SPLINE
SPL {X  -119.703, Y  +777.650, Z    +0.000, E1   -51.831, E3 +109843.279}
SPL {X  -145.184, Y  +738.720, Z    +0.000, E1   -43.488, E3 +109869.837}
SPL {X  -156.175, Y  +706.232, Z    +0.000, E1   -28.819, E3 +109878.722}
SPL {X  -159.337, Y  +685.942, Z    +0.000, E1   -14.672, E3 +109881.273}
SPL {X  -159.962, Y  +674.468, Z    +0.000, E1    -4.846, E3 +109881.892}
SPL {X  -159.990, Y  +669.479, Z    +0.000, E1    +0.004, E3 +109881.966}
SPL {X  -159.990, Y  +667.035, Z    +0.000, E1    +4.539, E3 +109881.997}
SPL {X  -159.990, Y  +662.914, Z    +0.000, E1   +13.494, E3 +109882.135}
SPL {X  -159.990, Y  +658.254, Z    +0.000, E1   +24.153, E3 +109882.413}
SPL {X  -159.990, Y  +652.944, Z    +0.000, E1   +35.122, E3 +109882.917}
SPL {X  -159.990, Y  +642.509, Z    +0.000, E1   +50.090, E3 +109884.488}
SPL {X  -159.990, Y  +618.566, Z    +0.000, E1   +64.119, E3 +109890.659}
SPL {X  -159.990, Y  +584.545, Z    +0.000, E1   +69.188, E3 +109903.194}
SPL {X  -159.990, Y  +578.002, Z    +0.000, E1   +69.607, E3 +109905.918}
SPL {X  -159.990, Y  +426.570, Z    +0.000, E1   +71.599, E3 +109986.408}
SPL {X  -159.990, Y  +405.946, Z    +0.000, E1   +71.630, E3 +110000.838}
SPL {X  -159.967, Y  +379.776, Z    +0.000, E1   +71.634, E3 +110019.284}
SPL {X  -158.535, Y  +360.970, Z    +0.000, E1   +71.460, E3 +110034.106}
SPL {X  -156.277, Y  +348.230, Z    +0.000, E1   +71.211, E3 +110045.450}
SPL {X  -155.351, Y  +344.251, Z    +0.000, E1   +70.004, E3 +110059.241}
SPL {X  -150.579, Y  +328.438, Z    +0.000, E1   +70.374, E3 +110067.627}
SPL {X  -146.933, Y  +319.195, Z    +0.000, E1   +70.230, E3 +110075.318}
SPL {X  -143.573, Y  +311.906, Z    +0.000, E1   +69.806, E3 +110083.628}
SPL {X  -139.693, Y  +304.508, Z    +0.000, E1   +69.301, E3 +110092.356}
SPL {X  -135.622, Y  +297.627, Z    +0.000, E1   +68.731, E3 +110100.764}
SPL {X  -131.165, Y  +290.889, Z    +0.000, E1   +68.094, E3 +110109.150}
SPL {X  -126.457, Y  +284.492, Z    +0.000, E1   +67.352, E3 +110117.235}
SPL {X  -123.432, Y  +280.710, Z    +0.000, E1   +66.830, E3 +110122.021}
SPL {X   -85.607, Y  +247.340, Z    +0.000, E1   +53.917, E3 +110263.742}
ENDSPLINE

SPLINE
SPL {X  -134.737, Y  +296.229, Z    +0.000, E1   +47.890, E3 +110406.515}
SPL {X  -154.917, Y  +342.531, Z    +0.000, E1   +31.203, E3 +110425.083}
SPL {X  -159.440, Y  +369.246, Z    +0.000, E1   +13.458, E3 +110428.982}
SPL {X  -159.987, Y  +381.470, Z    +0.000, E1    +2.976, E3 +110429.581}
SPL {X  -159.990, Y  +384.500, Z    +0.000, E1    +0.000, E3 +110429.614}
SPL {X  -159.990, Y  +386.323, Z    +0.000, E1    -3.079, E3 +110429.636}
SPL {X  -159.990, Y  +390.285, Z    +0.000, E1   -11.315, E3 +110429.757}
SPL {X  -159.990, Y  +394.559, Z    +0.000, E1   -20.770, E3 +110430.019}
SPL {X  -159.990, Y  +402.118, Z    +0.000, E1   -35.793, E3 +110430.810}
SPL {X  -159.990, Y  +415.193, Z    +0.000, E1   -52.724, E3 +110433.063}
SPL {X  -159.990, Y  +465.395, Z    +0.000, E1   -68.959, E3 +110448.152}
SPL {X  -159.990, Y  +657.157, Z    +0.000, E1   -72.499, E3 +110544.548}
SPL {X  -159.693, Y  +681.249, Z    +0.000, E1   -72.488, E3 +110560.942}
SPL {X  -157.599, Y  +699.059, Z    +0.000, E1   -72.249, E3 +110575.102}
SPL {X  -155.217, Y  +710.289, Z    +0.000, E1   -71.989, E3 +110585.119}
SPL {X  -152.611, Y  +719.527, Z    +0.000, E1   -71.702, E3 +110593.940}
SPL {X  -149.536, Y  +728.383, Z    +0.000, E1   -71.359, E3 +110602.919}
SPL {X  -146.250, Y  +736.367, Z    +0.000, E1   -70.965, E3 +110611.473}
SPL {X  -143.481, Y  +742.281, Z    +0.000, E1   -70.623, E3 +110618.069}
SPL {X  -140.071, Y  +748.811, Z    +0.000, E1   -70.193, E3 +110625.580}
SPL {X  -136.578, Y  +754.826, Z    +0.000, E1   -69.723, E3 +110632.710}
SPL {X  -133.265, Y  +760.028, Z    +0.000, E1   -69.258, E3 +110639.011}
SPL {X  -129.890, Y  +764.909, Z    +0.000, E1   -68.775, E3 +110644.981}
SPL {X  -125.802, Y  +770.346, Z    +0.000, E1   -68.156, E3 +110651.681}
SPL {X  -122.624, Y  +774.263, Z    +0.000, E1   -67.622, E3 +110656.503}
SPL {X   -84.435, Y  +807.395, Z    +0.000, E1   -55.948, E3 +110767.508}
ENDSPLINE

SPLINE
SPL {X  -119.703, Y  +777.650, Z    +0.000, E1   -51.831, E3 +110931.514}
SPL {X  -145.184, Y  +738.720, Z    +0.000, E1   -43.488, E3 +110958.072}
SPL {X  -154.467, Y  +713.173, Z    +0.000, E1   -32.658, E3 +110965.668}
SPL {X  -157.530, Y  +699.446, Z    +0.000, E1   -24.482, E3 +110968.084}
SPL {X  -159.337, Y  +685.942, Z    +0.000, E1   -14.672, E3 +110969.508}
SPL {X  -159.962, Y  +674.468, Z    +0.000, E1    -4.846, E3 +110970.127}
SPL {X  -159.990, Y  +669.479, Z    +0.000, E1    +0.004, E3 +110970.201}
SPL {X  -159.990, Y  +667.035, Z    +0.000, E1    +4.539, E3 +110970.232}
SPL {X  -159.990, Y  +662.914, Z    +0.000, E1   +13.494, E3 +110970.371}
SPL {X  -159.990, Y  +658.254, Z    +0.000, E1   +24.153, E3 +110970.648}
SPL {X  -159.990, Y  +652.944, Z    +0.000, E1   +35.122, E3 +110971.152}
SPL {X  -159.990, Y  +642.509, Z    +0.000, E1   +50.090, E3 +110972.724}
SPL {X  -159.990, Y  +618.566, Z    +0.000, E1   +64.119, E3 +110978.894}
SPL {X  -159.990, Y  +582.261, Z    +0.000, E1   +69.343, E3 +110992.380}
SPL {X  -159.990, Y  +406.555, Z    +0.000, E1   +71.635, E3 +111088.627}
SPL {X  -159.967, Y  +379.776, Z    +0.000, E1   +71.634, E3 +111107.520}
SPL {X  -158.535, Y  +360.970, Z    +0.000, E1   +71.460, E3 +111122.342}
SPL {X  -156.882, Y  +351.118, Z    +0.000, E1   +71.263, E3 +111131.053}
SPL {X  -155.538, Y  +345.018, Z    +0.000, E1   +71.109, E3 +111136.760}
SPL {X  -155.351, Y  +344.251, Z    +0.000, E1   +70.004, E3 +111147.477}
SPL {X  -150.579, Y  +328.438, Z    +0.000, E1   +70.374, E3 +111155.862}
SPL {X  -146.933, Y  +319.195, Z    +0.000, E1   +70.230, E3 +111163.553}
SPL {X  -143.573, Y  +311.906, Z    +0.000, E1   +69.806, E3 +111171.863}
SPL {X  -140.547, Y  +306.057, Z    +0.000, E1   +69.399, E3 +111178.755}
SPL {X  -137.438, Y  +300.600, Z    +0.000, E1   +68.984, E3 +111185.350}
SPL {X  -133.397, Y  +294.172, Z    +0.000, E1   +68.416, E3 +111193.285}
SPL {X  -128.822, Y  +287.623, Z    +0.000, E1   +67.729, E3 +111201.509}
SPL {X  -124.502, Y  +282.021, Z    +0.000, E1   +67.035, E3 +111208.583}
SPL {X   -85.607, Y  +247.340, Z    +0.000, E1   +53.917, E3 +111351.978}
ENDSPLINE

SPLINE
SPL {X  -134.737, Y  +296.229, Z    +0.000, E1   +47.890, E3 +111494.750}
SPL {X  -154.917, Y  +342.531, Z    +0.000, E1   +31.203, E3 +111513.318}
SPL {X  -159.440, Y  +369.246, Z    +0.000, E1   +13.458, E3 +111517.217}
SPL {X  -159.957, Y  +379.264, Z    +0.000, E1    +4.909, E3 +111517.773}
SPL {X  -159.990, Y  +384.398, Z    +0.000, E1    +0.172, E3 +111517.849}
SPL {X  -159.990, Y  +386.323, Z    +0.000, E1    -3.079, E3 +111517.871}
SPL {X  -159.990, Y  +390.285, Z    +0.000, E1   -11.315, E3 +111517.992}
SPL {X  -159.990, Y  +394.559, Z    +0.000, E1   -20.770, E3 +111518.254}
SPL {X  -159.990, Y  +402.118, Z    +0.000, E1   -35.793, E3 +111519.046}
SPL {X  -159.990, Y  +415.193, Z    +0.000, E1   -52.724, E3 +111521.298}
SPL {X  -159.990, Y  +465.395, Z    +0.000, E1   -68.959, E3 +111536.387}
SPL {X  -159.990, Y  +657.157, Z    +0.000, E1   -72.499, E3 +111632.784}
SPL {X  -159.947, Y  +675.227, Z    +0.000, E1   -72.487, E3 +111644.944}
SPL {X  -159.251, Y  +686.856, Z    +0.000, E1   -72.412, E3 +111653.472}
SPL {X  -157.599, Y  +699.059, Z    +0.000, E1   -72.249, E3 +111663.337}
SPL {X  -155.217, Y  +710.289, Z    +0.000, E1   -71.989, E3 +111673.354}
SPL {X  -152.611, Y  +719.527, Z    +0.000, E1   -71.702, E3 +111682.175}
SPL {X  -149.536, Y  +728.383, Z    +0.000, E1   -71.359, E3 +111691.154}
SPL {X  -146.250, Y  +736.367, Z    +0.000, E1   -70.965, E3 +111699.709}
SPL {X  -143.481, Y  +742.281, Z    +0.000, E1   -70.623, E3 +111706.304}
SPL {X  -140.071, Y  +748.811, Z    +0.000, E1   -70.193, E3 +111713.816}
SPL {X  -136.578, Y  +754.826, Z    +0.000, E1   -69.723, E3 +111720.945}
SPL {X  -133.265, Y  +760.028, Z    +0.000, E1   -69.258, E3 +111727.246}
SPL {X  -130.837, Y  +763.579, Z    +0.000, E1   -68.898, E3 +111731.606}
SPL {X  -127.941, Y  +767.561, Z    +0.000, E1   -68.475, E3 +111736.496}
SPL {X  -123.778, Y  +772.869, Z    +0.000, E1   -67.843, E3 +111743.004}
SPL {X   -84.435, Y  +807.395, Z    +0.000, E1   -55.948, E3 +111855.743}
ENDSPLINE

SPLINE
SPL {X  -119.703, Y  +777.650, Z    +0.000, E1   -51.831, E3 +112019.750}
SPL {X  -145.184, Y  +738.720, Z    +0.000, E1   -43.488, E3 +112046.308}
SPL {X  -154.467, Y  +713.173, Z    +0.000, E1   -32.658, E3 +112053.903}
SPL {X  -157.530, Y  +699.446, Z    +0.000, E1   -24.482, E3 +112056.319}
SPL {X  -159.337, Y  +685.942, Z    +0.000, E1   -14.672, E3 +112057.744}
SPL {X  -159.962, Y  +674.468, Z    +0.000, E1    -4.846, E3 +112058.362}
SPL {X  -159.990, Y  +669.479, Z    +0.000, E1    +0.004, E3 +112058.436}
SPL {X  -159.990, Y  +667.035, Z    +0.000, E1    +4.539, E3 +112058.467}
SPL {X  -159.990, Y  +662.914, Z    +0.000, E1   +13.494, E3 +112058.606}
SPL {X  -159.990, Y  +658.254, Z    +0.000, E1   +24.153, E3 +112058.884}
SPL {X  -159.990, Y  +652.944, Z    +0.000, E1   +35.122, E3 +112059.387}
SPL {X  -159.990, Y  +642.509, Z    +0.000, E1   +50.090, E3 +112060.959}
SPL {X  -159.990, Y  +618.566, Z    +0.000, E1   +64.119, E3 +112067.130}
SPL {X  -159.990, Y  +582.261, Z    +0.000, E1   +69.343, E3 +112080.615}
SPL {X  -159.990, Y  +406.555, Z    +0.000, E1   +71.635, E3 +112176.862}
SPL {X  -159.990, Y  +385.723, Z    +0.000, E1   +71.610, E3 +112191.600}
SPL {X  -159.404, Y  +368.814, Z    +0.000, E1   +71.556, E3 +112204.129}
SPL {X  -158.061, Y  +357.731, Z    +0.000, E1   +71.393, E3 +112213.397}
SPL {X  -156.277, Y  +348.230, Z    +0.000, E1   +71.211, E3 +112221.920}
SPL {X  -155.351, Y  +344.251, Z    +0.000, E1   +70.004, E3 +112235.712}
SPL {X  -150.579, Y  +328.438, Z    +0.000, E1   +70.374, E3 +112244.097}
SPL {X  -146.933, Y  +319.195, Z    +0.000, E1   +70.230, E3 +112251.788}
SPL {X  -143.573, Y  +311.906, Z    +0.000, E1   +69.806, E3 +112260.099}
SPL {X  -140.547, Y  +306.057, Z    +0.000, E1   +69.399, E3 +112266.991}
SPL {X  -137.438, Y  +300.600, Z    +0.000, E1   +68.984, E3 +112273.585}
SPL {X  -133.397, Y  +294.172, Z    +0.000, E1   +68.416, E3 +112281.520}
SPL {X  -128.822, Y  +287.623, Z    +0.000, E1   +67.729, E3 +112289.744}
SPL {X  -124.502, Y  +282.021, Z    +0.000, E1   +67.035, E3 +112296.818}
SPL {X   -85.607, Y  +247.340, Z    +0.000, E1   +53.917, E3 +112440.213}
ENDSPLINE

SPLINE
SPL {X  -134.737, Y  +296.229, Z    +0.000, E1   +47.890, E3 +112582.986}
SPL {X  -153.211, Y  +336.421, Z    +0.000, E1   +34.262, E3 +112600.194}
SPL {X  -158.240, Y  +358.900, Z    +0.000, E1   +21.089, E3 +112604.399}
SPL {X  -159.674, Y  +372.451, Z    +0.000, E1   +10.778, E3 +112605.695}
SPL {X  -159.987, Y  +381.470, Z    +0.000, E1    +2.976, E3 +112606.052}
SPL {X  -159.990, Y  +384.761, Z    +0.000, E1    -0.257, E3 +112606.087}
SPL {X  -159.990, Y  +389.248, Z    +0.000, E1    -8.879, E3 +112606.191}
SPL {X  -159.990, Y  +394.559, Z    +0.000, E1   -20.770, E3 +112606.490}
SPL {X  -159.990, Y  +402.118, Z    +0.000, E1   -35.793, E3 +112607.281}
SPL {X  -159.990, Y  +415.193, Z    +0.000, E1   -52.724, E3 +112609.534}
SPL {X  -159.990, Y  +465.395, Z    +0.000, E1   -68.959, E3 +112624.622}
SPL {X  -159.990, Y  +657.157, Z    +0.000, E1   -72.499, E3 +112721.019}
SPL {X  -159.693, Y  +681.249, Z    +0.000, E1   -72.488, E3 +112737.413}
SPL {X  -157.599, Y  +699.059, Z    +0.000, E1   -72.249, E3 +112751.573}
SPL {X  -155.217, Y  +710.289, Z    +0.000, E1   -71.989, E3 +112761.589}
SPL {X  -152.611, Y  +719.527, Z    +0.000, E1   -71.702, E3 +112770.410}
SPL {X  -149.536, Y  +728.383, Z    +0.000, E1   -71.359, E3 +112779.390}
SPL {X  -146.250, Y  +736.367, Z    +0.000, E1   -70.965, E3 +112787.944}
SPL {X  -143.481, Y  +742.281, Z    +0.000, E1   -70.623, E3 +112794.539}
SPL {X  -140.071, Y  +748.811, Z    +0.000, E1   -70.193, E3 +112802.051}
SPL {X  -136.578, Y  +754.826, Z    +0.000, E1   -69.723, E3 +112809.180}
SPL {X  -133.265, Y  +760.028, Z    +0.000, E1   -69.258, E3 +112815.481}
SPL {X  -130.837, Y  +763.579, Z    +0.000, E1   -68.898, E3 +112819.841}
SPL {X  -127.941, Y  +767.561, Z    +0.000, E1   -68.475, E3 +112824.732}
SPL {X  -123.778, Y  +772.869, Z    +0.000, E1   -67.843, E3 +112831.239}
SPL {X   -84.435, Y  +807.395, Z    +0.000, E1   -55.948, E3 +112943.978}
ENDSPLINE

SPLINE
SPL {X  -119.703, Y  +777.650, Z    +0.000, E1   -51.831, E3 +113107.985}
SPL {X  -145.184, Y  +738.720, Z    +0.000, E1   -43.488, E3 +113134.543}
SPL {X  -156.175, Y  +706.232, Z    +0.000, E1   -28.819, E3 +113143.428}
SPL {X  -159.337, Y  +685.942, Z    +0.000, E1   -14.672, E3 +113145.979}
SPL {X  -159.900, Y  +676.871, Z    +0.000, E1    -6.955, E3 +113146.527}
SPL {X  -159.990, Y  +669.634, Z    +0.000, E1    -0.285, E3 +113146.670}
SPL {X  -159.990, Y  +667.035, Z    +0.000, E1    +4.539, E3 +113146.702}
SPL {X  -159.990, Y  +662.914, Z    +0.000, E1   +13.494, E3 +113146.841}
SPL {X  -159.990, Y  +658.254, Z    +0.000, E1   +24.153, E3 +113147.119}
SPL {X  -159.990, Y  +652.944, Z    +0.000, E1   +35.122, E3 +113147.623}
SPL {X  -159.990, Y  +642.509, Z    +0.000, E1   +50.090, E3 +113149.194}
SPL {X  -159.990, Y  +618.566, Z    +0.000, E1   +64.119, E3 +113155.365}
SPL {X  -159.990, Y  +584.545, Z    +0.000, E1   +69.188, E3 +113167.900}
SPL {X  -159.990, Y  +578.002, Z    +0.000, E1   +69.607, E3 +113170.624}
SPL {X  -159.990, Y  +426.570, Z    +0.000, E1   +71.599, E3 +113251.114}
SPL {X  -159.990, Y  +405.946, Z    +0.000, E1   +71.630, E3 +113265.544}
SPL {X  -159.967, Y  +379.776, Z    +0.000, E1   +71.634, E3 +113283.990}
SPL {X  -158.535, Y  +360.970, Z    +0.000, E1   +71.460, E3 +113298.812}
SPL {X  -156.277, Y  +348.230, Z    +0.000, E1   +71.211, E3 +113310.155}
SPL {X  -155.351, Y  +344.251, Z    +0.000, E1   +70.004, E3 +113323.947}
SPL {X  -150.579, Y  +328.438, Z    +0.000, E1   +70.374, E3 +113332.333}
SPL {X  -146.933, Y  +319.195, Z    +0.000, E1   +70.230, E3 +113340.024}
SPL {X  -143.573, Y  +311.906, Z    +0.000, E1   +69.806, E3 +113348.334}
SPL {X  -140.547, Y  +306.057, Z    +0.000, E1   +69.399, E3 +113355.226}
SPL {X  -137.438, Y  +300.600, Z    +0.000, E1   +68.984, E3 +113361.820}
SPL {X  -133.397, Y  +294.172, Z    +0.000, E1   +68.416, E3 +113369.755}
SPL {X  -129.981, Y  +289.217, Z    +0.000, E1   +67.880, E3 +113376.005}
SPL {X  -126.457, Y  +284.492, Z    +0.000, E1   +67.352, E3 +113381.941}
SPL {X  -123.432, Y  +280.710, Z    +0.000, E1   +66.830, E3 +113386.727}
SPL {X   -85.607, Y  +247.340, Z    +0.000, E1   +53.917, E3 +113528.448}
ENDSPLINE

SPLINE
SPL {X  -119.557, Y  +276.184, Z    +0.000, E1   +51.032, E3 +113651.985}
SPL {X  -138.294, Y  +302.054, Z    +0.000, E1   +46.576, E3 +113675.307}
SPL {X  -153.211, Y  +336.421, Z    +0.000, E1   +34.262, E3 +113688.429}
SPL {X  -158.240, Y  +358.900, Z    +0.000, E1   +21.089, E3 +113692.634}
SPL {X  -159.854, Y  +375.896, Z    +0.000, E1    +7.981, E3 +113694.100}
SPL {X  -159.990, Y  +384.398, Z    +0.000, E1    +0.172, E3 +113694.320}
SPL {X  -159.990, Y  +386.323, Z    +0.000, E1    -3.079, E3 +113694.342}
SPL {X  -159.990, Y  +390.285, Z    +0.000, E1   -11.315, E3 +113694.463}
SPL {X  -159.990, Y  +394.559, Z    +0.000, E1   -20.770, E3 +113694.725}
SPL {X  -159.990, Y  +402.118, Z    +0.000, E1   -35.793, E3 +113695.516}
SPL {X  -159.990, Y  +415.193, Z    +0.000, E1   -52.724, E3 +113697.769}
SPL {X  -159.990, Y  +465.395, Z    +0.000, E1   -68.959, E3 +113712.857}
SPL {X  -159.990, Y  +657.157, Z    +0.000, E1   -72.499, E3 +113809.254}
SPL {X  -159.693, Y  +681.249, Z    +0.000, E1   -72.488, E3 +113825.648}
SPL {X  -157.599, Y  +699.059, Z    +0.000, E1   -72.249, E3 +113839.808}
SPL {X  -155.217, Y  +710.289, Z    +0.000, E1   -71.989, E3 +113849.825}
SPL {X  -152.611, Y  +719.527, Z    +0.000, E1   -71.702, E3 +113858.646}
SPL {X  -149.536, Y  +728.383, Z    +0.000, E1   -71.359, E3 +113867.625}
SPL {X  -146.250, Y  +736.367, Z    +0.000, E1   -70.965, E3 +113876.179}
SPL {X  -143.481, Y  +742.281, Z    +0.000, E1   -70.623, E3 +113882.775}
SPL {X  -140.071, Y  +748.811, Z    +0.000, E1   -70.193, E3 +113890.286}
SPL {X  -136.578, Y  +754.826, Z    +0.000, E1   -69.723, E3 +113897.416}
SPL {X  -133.265, Y  +760.028, Z    +0.000, E1   -69.258, E3 +113903.717}
SPL {X  -129.890, Y  +764.909, Z    +0.000, E1   -68.775, E3 +113909.687}
SPL {X  -125.802, Y  +770.346, Z    +0.000, E1   -68.156, E3 +113916.386}
SPL {X  -122.624, Y  +774.263, Z    +0.000, E1   -67.622, E3 +113921.209}
SPL {X   -84.435, Y  +807.395, Z    +0.000, E1   -55.948, E3 +114032.214}
ENDSPLINE

SPLINE
SPL {X  -119.703, Y  +777.650, Z    +0.000, E1   -51.831, E3 +114196.220}
SPL {X  -145.184, Y  +738.720, Z    +0.000, E1   -43.488, E3 +114222.778}
SPL {X  -154.467, Y  +713.173, Z    +0.000, E1   -32.658, E3 +114230.374}
SPL {X  -157.530, Y  +699.446, Z    +0.000, E1   -24.482, E3 +114232.789}
SPL {X  -159.337, Y  +685.942, Z    +0.000, E1   -14.672, E3 +114234.214}
SPL {X  -159.900, Y  +676.871, Z    +0.000, E1    -6.955, E3 +114234.762}
SPL {X  -159.990, Y  +669.634, Z    +0.000, E1    -0.285, E3 +114234.906}
SPL {X  -159.990, Y  +667.035, Z    +0.000, E1    +4.539, E3 +114234.938}
SPL {X  -159.990, Y  +662.914, Z    +0.000, E1   +13.494, E3 +114235.077}
SPL {X  -159.990, Y  +658.254, Z    +0.000, E1   +24.153, E3 +114235.354}
SPL {X  -159.990, Y  +650.381, Z    +0.000, E1   +39.393, E3 +114236.206}
SPL {X  -159.990, Y  +638.701, Z    +0.000, E1   +53.953, E3 +114238.092}
SPL {X  -159.990, Y  +618.566, Z    +0.000, E1   +64.119, E3 +114243.600}
SPL {X  -159.990, Y  +582.261, Z    +0.000, E1   +69.343, E3 +114257.086}
SPL {X  -159.990, Y  +406.555, Z    +0.000, E1   +71.635, E3 +114353.332}
SPL {X  -159.990, Y  +385.723, Z    +0.000, E1   +71.610, E3 +114368.071}
SPL {X  -159.404, Y  +368.814, Z    +0.000, E1   +71.556, E3 +114380.600}
SPL {X  -158.061, Y  +357.731, Z    +0.000, E1   +71.393, E3 +114389.868}
SPL {X  -156.277, Y  +348.230, Z    +0.000, E1   +71.211, E3 +114398.391}
SPL {X  -155.351, Y  +344.251, Z    +0.000, E1   +70.004, E3 +114412.183}
SPL {X  -150.579, Y  +328.438, Z    +0.000, E1   +70.374, E3 +114420.568}
SPL {X  -146.933, Y  +319.195, Z    +0.000, E1   +70.230, E3 +114428.259}
SPL {X  -143.573, Y  +311.906, Z    +0.000, E1   +69.806, E3 +114436.569}
SPL {X  -140.547, Y  +306.057, Z    +0.000, E1   +69.399, E3 +114443.461}
SPL {X  -137.438, Y  +300.600, Z    +0.000, E1   +68.984, E3 +114450.056}
SPL {X  -133.397, Y  +294.172, Z    +0.000, E1   +68.416, E3 +114457.990}
SPL {X  -128.822, Y  +287.623, Z    +0.000, E1   +67.729, E3 +114466.215}
SPL {X  -124.502, Y  +282.021, Z    +0.000, E1   +67.035, E3 +114473.289}
SPL {X   -85.607, Y  +247.340, Z    +0.000, E1   +53.917, E3 +114616.683}
ENDSPLINE

SPLINE
SPL {X  -134.737, Y  +296.229, Z    +0.000, E1   +47.890, E3 +114759.456}
SPL {X  -154.917, Y  +342.531, Z    +0.000, E1   +31.203, E3 +114778.024}
SPL {X  -159.440, Y  +369.246, Z    +0.000, E1   +13.458, E3 +114781.923}
SPL {X  -159.987, Y  +381.470, Z    +0.000, E1    +2.976, E3 +114782.522}
SPL {X  -159.990, Y  +384.500, Z    +0.000, E1    +0.000, E3 +114782.555}
SPL {X  -159.990, Y  +386.323, Z    +0.000, E1    -3.079, E3 +114782.577}
SPL {X  -159.990, Y  +390.285, Z    +0.000, E1   -11.315, E3 +114782.698}
SPL {X  -159.990, Y  +394.559, Z    +0.000, E1   -20.770, E3 +114782.960}
SPL {X  -159.990, Y  +399.334, Z    +0.000, E1   -30.876, E3 +114783.399}
SPL {X  -159.990, Y  +405.006, Z    +0.000, E1   -40.810, E3 +114784.117}
SPL {X  -159.990, Y  +415.193, Z    +0.000, E1   -52.724, E3 +114786.004}
SPL {X  -159.990, Y  +465.395, Z    +0.000, E1   -68.959, E3 +114801.093}
SPL {X  -159.990, Y  +657.157, Z    +0.000, E1   -72.499, E3 +114897.490}
SPL {X  -159.693, Y  +681.249, Z    +0.000, E1   -72.488, E3 +114913.884}
SPL {X  -157.599, Y  +699.059, Z    +0.000, E1   -72.249, E3 +114928.043}
SPL {X  -155.217, Y  +710.289, Z    +0.000, E1   -71.989, E3 +114938.060}
SPL {X  -152.611, Y  +719.527, Z    +0.000, E1   -71.702, E3 +114946.881}
SPL {X  -149.536, Y  +728.383, Z    +0.000, E1   -71.359, E3 +114955.860}
SPL {X  -146.250, Y  +736.367, Z    +0.000, E1   -70.965, E3 +114964.414}
SPL {X  -143.481, Y  +742.281, Z    +0.000, E1   -70.623, E3 +114971.010}
SPL {X  -140.071, Y  +748.811, Z    +0.000, E1   -70.193, E3 +114978.522}
SPL {X  -136.578, Y  +754.826, Z    +0.000, E1   -69.723, E3 +114985.651}
SPL {X  -133.265, Y  +760.028, Z    +0.000, E1   -69.258, E3 +114991.952}
SPL {X  -130.837, Y  +763.579, Z    +0.000, E1   -68.898, E3 +114996.312}
SPL {X  -127.941, Y  +767.561, Z    +0.000, E1   -68.475, E3 +115001.202}
SPL {X  -123.778, Y  +772.869, Z    +0.000, E1   -67.843, E3 +115007.710}
SPL {X   -84.435, Y  +807.395, Z    +0.000, E1   -55.948, E3 +115120.449}
ENDSPLINE

SPLINE
SPL {X  -119.703, Y  +777.650, Z    +0.000, E1   -51.831, E3 +115284.455}
SPL {X  -145.184, Y  +738.720, Z    +0.000, E1   -43.488, E3 +115311.013}
SPL {X  -156.175, Y  +706.232, Z    +0.000, E1   -28.819, E3 +115319.898}
SPL {X  -159.337, Y  +685.942, Z    +0.000, E1   -14.672, E3 +115322.449}
SPL {X  -159.962, Y  +674.468, Z    +0.000, E1    -4.846, E3 +115323.068}
SPL {X  -159.990, Y  +669.479, Z    +0.000, E1    +0.004, E3 +115323.142}
SPL {X  -159.990, Y  +667.035, Z    +0.000, E1    +4.539, E3 +115323.173}
SPL {X  -159.990, Y  +662.914, Z    +0.000, E1   +13.494, E3 +115323.312}
SPL {X  -159.990, Y  +658.254, Z    +0.000, E1   +24.153, E3 +115323.590}
SPL {X  -159.990, Y  +652.944, Z    +0.000, E1   +35.122, E3 +115324.093}
SPL {X  -159.990, Y  +642.509, Z    +0.000, E1   +50.090, E3 +115325.665}
SPL {X  -159.990, Y  +618.566, Z    +0.000, E1   +64.119, E3 +115331.835}
SPL {X  -159.990, Y  +584.545, Z    +0.000, E1   +69.188, E3 +115344.371}
SPL {X  -159.990, Y  +578.002, Z    +0.000, E1   +69.607, E3 +115347.094}
SPL {X  -159.990, Y  +426.570, Z    +0.000, E1   +71.599, E3 +115427.584}
SPL {X  -159.990, Y  +405.946, Z    +0.000, E1   +71.630, E3 +115442.014}
SPL {X  -159.967, Y  +379.776, Z    +0.000, E1   +71.634, E3 +115460.461}
SPL {X  -158.535, Y  +360.970, Z    +0.000, E1   +71.460, E3 +115475.283}
SPL {X  -156.882, Y  +351.118, Z    +0.000, E1   +71.263, E3 +115483.995}
SPL {X  -155.889, Y  +346.508, Z    +0.000, E1   +70.461, E3 +115494.857}
SPL {X  -154.332, Y  +340.328, Z    +0.000, E1   +70.024, E3 +115503.085}
SPL {X  -150.579, Y  +328.438, Z    +0.000, E1   +70.374, E3 +115508.803}
SPL {X  -146.933, Y  +319.195, Z    +0.000, E1   +70.230, E3 +115516.494}
SPL {X  -143.573, Y  +311.906, Z    +0.000, E1   +69.806, E3 +115524.805}
SPL {X  -139.693, Y  +304.508, Z    +0.000, E1   +69.301, E3 +115533.533}
SPL {X  -135.622, Y  +297.627, Z    +0.000, E1   +68.731, E3 +115541.941}
SPL {X  -131.165, Y  +290.889, Z    +0.000, E1   +68.094, E3 +115550.326}
SPL {X  -126.457, Y  +284.492, Z    +0.000, E1   +67.352, E3 +115558.412}
SPL {X  -123.432, Y  +280.710, Z    +0.000, E1   +66.830, E3 +115563.197}
SPL {X   -85.607, Y  +247.340, Z    +0.000, E1   +53.917, E3 +115704.919}
ENDSPLINE

SPLINE
SPL {X  -134.737, Y  +296.229, Z    +0.000, E1   +47.890, E3 +115847.692}
SPL {X  -154.917, Y  +342.531, Z    +0.000, E1   +31.203, E3 +115866.259}
SPL {X  -159.440, Y  +369.246, Z    +0.000, E1   +13.458, E3 +115870.159}
SPL {X  -159.987, Y  +381.470, Z    +0.000, E1    +2.976, E3 +115870.757}
SPL {X  -159.990, Y  +384.500, Z    +0.000, E1    +0.000, E3 +115870.791}
SPL {X  -159.990, Y  +386.323, Z    +0.000, E1    -3.079, E3 +115870.812}
SPL {X  -159.990, Y  +390.285, Z    +0.000, E1   -11.315, E3 +115870.933}
SPL {X  -159.990, Y  +394.559, Z    +0.000, E1   -20.770, E3 +115871.195}
SPL {X  -159.990, Y  +399.334, Z    +0.000, E1   -30.876, E3 +115871.634}
SPL {X  -159.990, Y  +405.006, Z    +0.000, E1   -40.810, E3 +115872.352}
SPL {X  -159.990, Y  +415.193, Z    +0.000, E1   -52.724, E3 +115874.239}
SPL {X  -159.990, Y  +465.395, Z    +0.000, E1   -68.959, E3 +115889.328}
SPL {X  -159.990, Y  +657.157, Z    +0.000, E1   -72.499, E3 +115985.725}
SPL {X  -159.693, Y  +681.249, Z    +0.000, E1   -72.488, E3 +116002.119}
SPL {X  -157.599, Y  +699.059, Z    +0.000, E1   -72.249, E3 +116016.278}
SPL {X  -155.217, Y  +710.289, Z    +0.000, E1   -71.989, E3 +116026.295}
SPL {X  -152.611, Y  +719.527, Z    +0.000, E1   -71.702, E3 +116035.116}
SPL {X  -149.536, Y  +728.383, Z    +0.000, E1   -71.359, E3 +116044.096}
SPL {X  -146.250, Y  +736.367, Z    +0.000, E1   -70.965, E3 +116052.650}
SPL {X  -143.481, Y  +742.281, Z    +0.000, E1   -70.623, E3 +116059.245}
SPL {X  -140.071, Y  +748.811, Z    +0.000, E1   -70.193, E3 +116066.757}
SPL {X  -136.578, Y  +754.826, Z    +0.000, E1   -69.723, E3 +116073.886}
SPL {X  -133.265, Y  +760.028, Z    +0.000, E1   -69.258, E3 +116080.187}
SPL {X  -130.837, Y  +763.579, Z    +0.000, E1   -68.898, E3 +116084.547}
SPL {X  -127.941, Y  +767.561, Z    +0.000, E1   -68.475, E3 +116089.438}
SPL {X  -123.778, Y  +772.869, Z    +0.000, E1   -67.843, E3 +116095.945}
SPL {X   -84.435, Y  +807.395, Z    +0.000, E1   -55.948, E3 +116208.684}
ENDSPLINE

SPLINE
SPL {X  -119.703, Y  +777.650, Z    +0.000, E1   -51.831, E3 +116372.691}
SPL {X  -145.184, Y  +738.720, Z    +0.000, E1   -43.488, E3 +116399.249}
SPL {X  -156.175, Y  +706.232, Z    +0.000, E1   -28.819, E3 +116408.134}
SPL {X  -159.337, Y  +685.942, Z    +0.000, E1   -14.672, E3 +116410.685}
SPL {X  -159.962, Y  +674.468, Z    +0.000, E1    -4.846, E3 +116411.303}
SPL {X  -159.990, Y  +669.479, Z    +0.000, E1    +0.004, E3 +116411.378}
SPL {X  -159.990, Y  +667.035, Z    +0.000, E1    +4.539, E3 +116411.408}
SPL {X  -159.990, Y  +662.914, Z    +0.000, E1   +13.494, E3 +116411.547}
SPL {X  -159.990, Y  +658.254, Z    +0.000, E1   +24.153, E3 +116411.825}
SPL {X  -159.990, Y  +652.944, Z    +0.000, E1   +35.122, E3 +116412.329}
SPL {X  -159.990, Y  +646.557, Z    +0.000, E1   +45.390, E3 +116413.195}
SPL {X  -159.990, Y  +638.701, Z    +0.000, E1   +53.953, E3 +116414.562}
SPL {X  -159.990, Y  +618.566, Z    +0.000, E1   +64.119, E3 +116420.071}
SPL {X  -159.990, Y  +582.261, Z    +0.000, E1   +69.343, E3 +116433.556}
SPL {X  -159.990, Y  +426.570, Z    +0.000, E1   +71.599, E3 +116515.820}
SPL {X  -159.990, Y  +405.946, Z    +0.000, E1   +71.630, E3 +116530.250}
SPL {X  -159.990, Y  +385.723, Z    +0.000, E1   +71.610, E3 +116544.541}
SPL {X  -159.404, Y  +368.814, Z    +0.000, E1   +71.556, E3 +116557.071}
SPL {X  -158.061, Y  +357.731, Z    +0.000, E1   +71.393, E3 +116566.338}
SPL {X  -156.277, Y  +348.230, Z    +0.000, E1   +71.211, E3 +116574.861}
SPL {X  -155.351, Y  +344.251, Z    +0.000, E1   +70.004, E3 +116588.653}
SPL {X  -150.579, Y  +328.438, Z    +0.000, E1   +70.374, E3 +116597.039}
SPL {X  -146.933, Y  +319.195, Z    +0.000, E1   +70.230, E3 +116604.730}
SPL {X  -143.573, Y  +311.906, Z    +0.000, E1   +69.806, E3 +116613.040}
SPL {X  -140.547, Y  +306.057, Z    +0.000, E1   +69.399, E3 +116619.932}
SPL {X  -136.400, Y  +298.883, Z    +0.000, E1   +68.867, E3 +116628.588}
SPL {X  -131.165, Y  +290.889, Z    +0.000, E1   +68.094, E3 +116638.562}
SPL {X  -126.457, Y  +284.492, Z    +0.000, E1   +67.352, E3 +116646.647}
SPL {X  -123.432, Y  +280.710, Z    +0.000, E1   +66.830, E3 +116651.433}
SPL {X   -85.607, Y  +247.340, Z    +0.000, E1   +53.917, E3 +116793.154}
ENDSPLINE

SPLINE
SPL {X  -119.557, Y  +276.184, Z    +0.000, E1   +51.032, E3 +116916.691}
SPL {X  -138.294, Y  +302.054, Z    +0.000, E1   +46.576, E3 +116940.013}
SPL {X  -153.211, Y  +336.421, Z    +0.000, E1   +34.262, E3 +116953.135}
SPL {X  -158.240, Y  +358.900, Z    +0.000, E1   +21.089, E3 +116957.340}
SPL {X  -159.674, Y  +372.451, Z    +0.000, E1   +10.778, E3 +116958.636}
SPL {X  -159.987, Y  +381.470, Z    +0.000, E1    +2.976, E3 +116958.993}
SPL {X  -159.990, Y  +384.761, Z    +0.000, E1    -0.257, E3 +116959.028}
SPL {X  -159.990, Y  +389.248, Z    +0.000, E1    -8.879, E3 +116959.132}
SPL {X  -159.990, Y  +394.559, Z    +0.000, E1   -20.770, E3 +116959.431}
SPL {X  -159.990, Y  +402.118, Z    +0.000, E1   -35.793, E3 +116960.222}
SPL {X  -159.990, Y  +415.193, Z    +0.000, E1   -52.724, E3 +116962.475}
SPL {X  -159.990, Y  +465.395, Z    +0.000, E1   -68.959, E3 +116977.563}
SPL {X  -159.990, Y  +657.157, Z    +0.000, E1   -72.499, E3 +117073.960}
SPL {X  -159.947, Y  +675.227, Z    +0.000, E1   -72.487, E3 +117086.120}
SPL {X  -159.251, Y  +686.856, Z    +0.000, E1   -72.412, E3 +117094.648}
SPL {X  -157.599, Y  +699.059, Z    +0.000, E1   -72.249, E3 +117104.514}
SPL {X  -155.217, Y  +710.289, Z    +0.000, E1   -71.989, E3 +117114.530}
SPL {X  -152.611, Y  +719.527, Z    +0.000, E1   -71.702, E3 +117123.352}
SPL {X  -149.536, Y  +728.383, Z    +0.000, E1   -71.359, E3 +117132.331}
SPL {X  -146.250, Y  +736.367, Z    +0.000, E1   -70.965, E3 +117140.885}
SPL {X  -143.481, Y  +742.281, Z    +0.000, E1   -70.623, E3 +117147.480}
SPL {X  -140.071, Y  +748.811, Z    +0.000, E1   -70.193, E3 +117154.992}
SPL {X  -136.578, Y  +754.826, Z    +0.000, E1   -69.723, E3 +117162.122}
SPL {X  -132.176, Y  +761.646, Z    +0.000, E1   -69.128, E3 +117170.365}
SPL {X  -127.941, Y  +767.561, Z    +0.000, E1   -68.475, E3 +117177.673}
SPL {X  -123.778, Y  +772.869, Z    +0.000, E1   -67.843, E3 +117184.180}
SPL {X   -84.435, Y  +807.395, Z    +0.000, E1   -55.948, E3 +117296.919}
ENDSPLINE

SPLINE
SPL {X  -119.703, Y  +777.650, Z    +0.000, E1   -51.831, E3 +117460.926}
SPL {X  -145.184, Y  +738.720, Z    +0.000, E1   -43.488, E3 +117487.484}
SPL {X  -156.175, Y  +706.232, Z    +0.000, E1   -28.819, E3 +117496.369}
SPL {X  -159.337, Y  +685.942, Z    +0.000, E1   -14.672, E3 +117498.920}
SPL {X  -159.900, Y  +676.871, Z    +0.000, E1    -6.955, E3 +117499.468}
SPL {X  -159.990, Y  +669.634, Z    +0.000, E1    -0.285, E3 +117499.612}
SPL {X  -159.990, Y  +667.035, Z    +0.000, E1    +4.539, E3 +117499.644}
SPL {X  -159.990, Y  +662.914, Z    +0.000, E1   +13.494, E3 +117499.782}
SPL {X  -159.990, Y  +658.254, Z    +0.000, E1   +24.153, E3 +117500.060}
SPL {X  -159.990, Y  +652.944, Z    +0.000, E1   +35.122, E3 +117500.564}
SPL {X  -159.990, Y  +646.557, Z    +0.000, E1   +45.390, E3 +117501.431}
SPL {X  -159.990, Y  +638.701, Z    +0.000, E1   +53.953, E3 +117502.798}
SPL {X  -159.990, Y  +618.566, Z    +0.000, E1   +64.119, E3 +117508.306}
SPL {X  -159.990, Y  +582.261, Z    +0.000, E1   +69.343, E3 +117521.792}
SPL {X  -159.990, Y  +426.570, Z    +0.000, E1   +71.599, E3 +117604.055}
SPL {X  -159.990, Y  +405.946, Z    +0.000, E1   +71.630, E3 +117618.485}
SPL {X  -159.990, Y  +385.723, Z    +0.000, E1   +71.610, E3 +117632.777}
SPL {X  -159.404, Y  +368.814, Z    +0.000, E1   +71.556, E3 +117645.306}
SPL {X  -158.061, Y  +357.731, Z    +0.000, E1   +71.393, E3 +117654.574}
SPL {X  -156.277, Y  +348.230, Z    +0.000, E1   +71.211, E3 +117663.097}
SPL {X  -155.351, Y  +344.251, Z    +0.000, E1   +70.004, E3 +117676.889}
SPL {X  -150.579, Y  +328.438, Z    +0.000, E1   +70.374, E3 +117685.274}
SPL {X  -146.933, Y  +319.195, Z    +0.000, E1   +70.230, E3 +117692.965}
SPL {X  -143.573, Y  +311.906, Z    +0.000, E1   +69.806, E3 +117701.275}
SPL {X  -140.547, Y  +306.057, Z    +0.000, E1   +69.399, E3 +117708.167}
SPL {X  -137.438, Y  +300.600, Z    +0.000, E1   +68.984, E3 +117714.761}
SPL {X  -133.397, Y  +294.172, Z    +0.000, E1   +68.416, E3 +117722.696}
SPL {X  -129.981, Y  +289.217, Z    +0.000, E1   +67.880, E3 +117728.946}
SPL {X  -126.457, Y  +284.492, Z    +0.000, E1   +67.352, E3 +117734.882}
SPL {X  -123.432, Y  +280.710, Z    +0.000, E1   +66.830, E3 +117739.668}
SPL {X   -85.607, Y  +247.340, Z    +0.000, E1   +53.917, E3 +117881.389}
ENDSPLINE

SPLINE
SPL {X  -119.557, Y  +276.184, Z    +0.000, E1   +51.032, E3 +118004.926}
SPL {X  -138.294, Y  +302.054, Z    +0.000, E1   +46.576, E3 +118028.248}
SPL {X  -153.211, Y  +336.421, Z    +0.000, E1   +34.262, E3 +118041.370}
SPL {X  -158.240, Y  +358.900, Z    +0.000, E1   +21.089, E3 +118045.575}
SPL {X  -159.674, Y  +372.451, Z    +0.000, E1   +10.778, E3 +118046.871}
SPL {X  -159.987, Y  +381.470, Z    +0.000, E1    +2.976, E3 +118047.228}
SPL {X  -159.990, Y  +384.500, Z    +0.000, E1    +0.000, E3 +118047.261}
SPL {X  -159.990, Y  +386.323, Z    +0.000, E1    -3.079, E3 +118047.283}
SPL {X  -159.990, Y  +390.285, Z    +0.000, E1   -11.315, E3 +118047.404}
SPL {X  -159.990, Y  +394.559, Z    +0.000, E1   -20.770, E3 +118047.666}
SPL {X  -159.990, Y  +399.334, Z    +0.000, E1   -30.876, E3 +118048.105}
SPL {X  -159.990, Y  +405.006, Z    +0.000, E1   -40.810, E3 +118048.823}
SPL {X  -159.990, Y  +415.193, Z    +0.000, E1   -52.724, E3 +118050.710}
SPL {X  -159.990, Y  +465.395, Z    +0.000, E1   -68.959, E3 +118065.799}
SPL {X  -159.990, Y  +652.170, Z    +0.000, E1   -72.485, E3 +118158.894}
SPL {X  -159.990, Y  +670.864, Z    +0.000, E1   -72.509, E3 +118171.342}
SPL {X  -159.251, Y  +686.856, Z    +0.000, E1   -72.412, E3 +118182.884}
SPL {X  -157.599, Y  +699.059, Z    +0.000, E1   -72.249, E3 +118192.749}
SPL {X  -155.217, Y  +710.289, Z    +0.000, E1   -71.989, E3 +118202.766}
SPL {X  -152.611, Y  +719.527, Z    +0.000, E1   -71.702, E3 +118211.587}
SPL {X  -149.536, Y  +728.383, Z    +0.000, E1   -71.359, E3 +118220.566}
SPL {X  -146.250, Y  +736.367, Z    +0.000, E1   -70.965, E3 +118229.120}
SPL {X  -143.481, Y  +742.281, Z    +0.000, E1   -70.623, E3 +118235.716}
SPL {X  -140.071, Y  +748.811, Z    +0.000, E1   -70.193, E3 +118243.227}
SPL {X  -136.578, Y  +754.826, Z    +0.000, E1   -69.723, E3 +118250.357}
SPL {X  -132.176, Y  +761.646, Z    +0.000, E1   -69.128, E3 +118258.600}
SPL {X  -127.941, Y  +767.561, Z    +0.000, E1   -68.475, E3 +118265.908}
SPL {X  -123.778, Y  +772.869, Z    +0.000, E1   -67.843, E3 +118272.416}
SPL {X   -84.435, Y  +807.395, Z    +0.000, E1   -55.948, E3 +118385.155}
ENDSPLINE

SPLINE
SPL {X  -119.703, Y  +777.650, Z    +0.000, E1   -51.831, E3 +118549.161}
SPL {X  -145.184, Y  +738.720, Z    +0.000, E1   -43.488, E3 +118575.719}
SPL {X  -156.175, Y  +706.232, Z    +0.000, E1   -28.819, E3 +118584.604}
SPL {X  -159.337, Y  +685.942, Z    +0.000, E1   -14.672, E3 +118587.155}
SPL {X  -159.900, Y  +676.871, Z    +0.000, E1    -6.955, E3 +118587.704}
SPL {X  -159.990, Y  +669.634, Z    +0.000, E1    -0.285, E3 +118587.847}
SPL {X  -159.990, Y  +667.035, Z    +0.000, E1    +4.539, E3 +118587.879}
SPL {X  -159.990, Y  +662.914, Z    +0.000, E1   +13.494, E3 +118588.018}
SPL {X  -159.990, Y  +658.254, Z    +0.000, E1   +24.153, E3 +118588.295}
SPL {X  -159.990, Y  +652.944, Z    +0.000, E1   +35.122, E3 +118588.799}
SPL {X  -159.990, Y  +642.509, Z    +0.000, E1   +50.090, E3 +118590.371}
SPL {X  -159.990, Y  +618.566, Z    +0.000, E1   +64.119, E3 +118596.541}
SPL {X  -159.990, Y  +582.261, Z    +0.000, E1   +69.343, E3 +118610.027}
SPL {X  -159.990, Y  +406.555, Z    +0.000, E1   +71.635, E3 +118706.274}
SPL {X  -159.990, Y  +385.723, Z    +0.000, E1   +71.610, E3 +118721.012}
SPL {X  -159.404, Y  +368.814, Z    +0.000, E1   +71.556, E3 +118733.541}
SPL {X  -157.440, Y  +354.048, Z    +0.000, E1   +71.342, E3 +118746.015}
SPL {X  -155.538, Y  +345.018, Z    +0.000, E1   +71.109, E3 +118754.407}
SPL {X  -155.351, Y  +344.251, Z    +0.000, E1   +70.004, E3 +118765.124}
SPL {X  -150.579, Y  +328.438, Z    +0.000, E1   +70.374, E3 +118773.509}
SPL {X  -146.933, Y  +319.195, Z    +0.000, E1   +70.230, E3 +118781.200}
SPL {X  -143.573, Y  +311.906, Z    +0.000, E1   +69.806, E3 +118789.510}
SPL {X  -140.547, Y  +306.057, Z    +0.000, E1   +69.399, E3 +118796.402}
SPL {X  -137.438, Y  +300.600, Z    +0.000, E1   +68.984, E3 +118802.997}
SPL {X  -133.397, Y  +294.172, Z    +0.000, E1   +68.416, E3 +118810.932}
SPL {X  -128.822, Y  +287.623, Z    +0.000, E1   +67.729, E3 +118819.156}
SPL {X  -124.502, Y  +282.021, Z    +0.000, E1   +67.035, E3 +118826.230}
SPL {X   -85.607, Y  +247.340, Z    +0.000, E1   +53.917, E3 +118969.625}
ENDSPLINE

SPLINE
SPL {X  -134.737, Y  +296.229, Z    +0.000, E1   +47.890, E3 +119112.398}
SPL {X  -154.917, Y  +342.531, Z    +0.000, E1   +31.203, E3 +119130.965}
SPL {X  -159.440, Y  +369.246, Z    +0.000, E1   +13.458, E3 +119134.864}
SPL {X  -159.957, Y  +379.264, Z    +0.000, E1    +4.909, E3 +119135.421}
SPL {X  -159.990, Y  +384.670, Z    +0.000, E1    -0.079, E3 +119135.498}
SPL {X  -159.990, Y  +389.248, Z    +0.000, E1    -8.879, E3 +119135.602}
SPL {X  -159.990, Y  +394.559, Z    +0.000, E1   -20.770, E3 +119135.901}
SPL {X  -159.990, Y  +402.118, Z    +0.000, E1   -35.793, E3 +119136.693}
SPL {X  -159.990, Y  +415.193, Z    +0.000, E1   -52.724, E3 +119138.945}
SPL {X  -159.990, Y  +465.395, Z    +0.000, E1   -68.959, E3 +119154.034}
SPL {X  -159.990, Y  +657.157, Z    +0.000, E1   -72.499, E3 +119250.431}
SPL {X  -159.693, Y  +681.249, Z    +0.000, E1   -72.488, E3 +119266.825}
SPL {X  -157.599, Y  +699.059, Z    +0.000, E1   -72.249, E3 +119280.984}
SPL {X  -155.217, Y  +710.289, Z    +0.000, E1   -71.989, E3 +119291.001}
SPL {X  -152.611, Y  +719.527, Z    +0.000, E1   -71.702, E3 +119299.822}
SPL {X  -149.536, Y  +728.383, Z    +0.000, E1   -71.359, E3 +119308.801}
SPL {X  -146.250, Y  +736.367, Z    +0.000, E1   -70.965, E3 +119317.356}
SPL {X  -143.481, Y  +742.281, Z    +0.000, E1   -70.623, E3 +119323.951}
SPL {X  -140.071, Y  +748.811, Z    +0.000, E1   -70.193, E3 +119331.463}
SPL {X  -136.578, Y  +754.826, Z    +0.000, E1   -69.723, E3 +119338.592}
SPL {X  -133.265, Y  +760.028, Z    +0.000, E1   -69.258, E3 +119344.893}
SPL {X  -129.890, Y  +764.909, Z    +0.000, E1   -68.775, E3 +119350.864}
SPL {X  -125.802, Y  +770.346, Z    +0.000, E1   -68.156, E3 +119357.563}
SPL {X  -122.624, Y  +774.263, Z    +0.000, E1   -67.622, E3 +119362.386}
SPL {X   -84.435, Y  +807.395, Z    +0.000, E1   -55.948, E3 +119473.390}
ENDSPLINE

SPLINE
SPL {X  -119.703, Y  +777.650, Z    +0.000, E1   -51.831, E3 +119637.397}
SPL {X  -145.184, Y  +738.720, Z    +0.000, E1   -43.488, E3 +119663.955}
SPL {X  -156.175, Y  +706.232, Z    +0.000, E1   -28.819, E3 +119672.839}
SPL {X  -159.337, Y  +685.942, Z    +0.000, E1   -14.672, E3 +119675.391}
SPL {X  -159.962, Y  +674.468, Z    +0.000, E1    -4.846, E3 +119676.009}
SPL {X  -159.990, Y  +669.479, Z    +0.000, E1    +0.004, E3 +119676.083}
SPL {X  -159.990, Y  +667.035, Z    +0.000, E1    +4.539, E3 +119676.114}
SPL {X  -159.990, Y  +662.914, Z    +0.000, E1   +13.494, E3 +119676.253}
SPL {X  -159.990, Y  +658.254, Z    +0.000, E1   +24.153, E3 +119676.531}
SPL {X  -159.990, Y  +652.944, Z    +0.000, E1   +35.122, E3 +119677.034}
SPL {X  -159.990, Y  +642.509, Z    +0.000, E1   +50.090, E3 +119678.606}
SPL {X  -159.990, Y  +618.566, Z    +0.000, E1   +64.119, E3 +119684.777}
SPL {X  -159.990, Y  +582.261, Z    +0.000, E1   +69.343, E3 +119698.262}
SPL {X  -159.990, Y  +406.555, Z    +0.000, E1   +71.635, E3 +119794.509}
SPL {X  -159.967, Y  +379.776, Z    +0.000, E1   +71.634, E3 +119813.402}
SPL {X  -158.535, Y  +360.970, Z    +0.000, E1   +71.460, E3 +119828.224}
SPL {X  -156.882, Y  +351.118, Z    +0.000, E1   +71.263, E3 +119836.936}
SPL {X  -155.538, Y  +345.018, Z    +0.000, E1   +71.109, E3 +119842.642}
SPL {X  -155.351, Y  +344.251, Z    +0.000, E1   +70.004, E3 +119853.359}
SPL {X  -150.579, Y  +328.438, Z    +0.000, E1   +70.374, E3 +119861.744}
SPL {X  -146.933, Y  +319.195, Z    +0.000, E1   +70.230, E3 +119869.435}
SPL {X  -143.573, Y  +311.906, Z    +0.000, E1   +69.806, E3 +119877.746}
SPL {X  -140.547, Y  +306.057, Z    +0.000, E1   +69.399, E3 +119884.638}
SPL {X  -136.400, Y  +298.883, Z    +0.000, E1   +68.867, E3 +119893.294}
SPL {X  -131.165, Y  +290.889, Z    +0.000, E1   +68.094, E3 +119903.267}
SPL {X  -126.457, Y  +284.492, Z    +0.000, E1   +67.352, E3 +119911.353}
SPL {X  -123.432, Y  +280.710, Z    +0.000, E1   +66.830, E3 +119916.139}
SPL {X   -85.607, Y  +247.340, Z    +0.000, E1   +53.917, E3 +120057.860}
ENDSPLINE

SPLINE
SPL {X  -134.737, Y  +296.229, Z    +0.000, E1   +47.890, E3 +120200.633}
SPL {X  -154.917, Y  +342.531, Z    +0.000, E1   +31.203, E3 +120219.200}
SPL {X  -159.440, Y  +369.246, Z    +0.000, E1   +13.458, E3 +120223.100}
SPL {X  -159.987, Y  +381.470, Z    +0.000, E1    +2.976, E3 +120223.699}
SPL {X  -159.990, Y  +384.761, Z    +0.000, E1    -0.257, E3 +120223.734}
SPL {X  -159.990, Y  +389.248, Z    +0.000, E1    -8.879, E3 +120223.838}
SPL {X  -159.990, Y  +394.559, Z    +0.000, E1   -20.770, E3 +120224.137}
SPL {X  -159.990, Y  +402.118, Z    +0.000, E1   -35.793, E3 +120224.928}
SPL {X  -159.990, Y  +415.193, Z    +0.000, E1   -52.724, E3 +120227.181}
SPL {X  -159.990, Y  +465.395, Z    +0.000, E1   -68.959, E3 +120242.269}
SPL {X  -159.990, Y  +657.157, Z    +0.000, E1   -72.499, E3 +120338.666}
SPL {X  -159.693, Y  +681.249, Z    +0.000, E1   -72.488, E3 +120355.060}
SPL {X  -157.599, Y  +699.059, Z    +0.000, E1   -72.249, E3 +120369.220}
SPL {X  -155.217, Y  +710.289, Z    +0.000, E1   -71.989, E3 +120379.236}
SPL {X  -152.611, Y  +719.527, Z    +0.000, E1   -71.702, E3 +120388.058}
SPL {X  -149.536, Y  +728.383, Z    +0.000, E1   -71.359, E3 +120397.037}
SPL {X  -146.250, Y  +736.367, Z    +0.000, E1   -70.965, E3 +120405.591}
SPL {X  -143.481, Y  +742.281, Z    +0.000, E1   -70.623, E3 +120412.186}
SPL {X  -140.071, Y  +748.811, Z    +0.000, E1   -70.193, E3 +120419.698}
SPL {X  -136.578, Y  +754.826, Z    +0.000, E1   -69.723, E3 +120426.827}
SPL {X  -133.265, Y  +760.028, Z    +0.000, E1   -69.258, E3 +120433.128}
SPL {X  -129.890, Y  +764.909, Z    +0.000, E1   -68.775, E3 +120439.099}
SPL {X  -125.802, Y  +770.346, Z    +0.000, E1   -68.156, E3 +120445.798}
SPL {X  -122.624, Y  +774.263, Z    +0.000, E1   -67.622, E3 +120450.621}
SPL {X   -84.435, Y  +807.395, Z    +0.000, E1   -55.948, E3 +120561.625}
ENDSPLINE

SPLINE
SPL {X  -119.703, Y  +777.650, Z    +0.000, E1   -51.831, E3 +120725.632}
SPL {X  -145.184, Y  +738.720, Z    +0.000, E1   -43.488, E3 +120752.190}
SPL {X  -154.467, Y  +713.173, Z    +0.000, E1   -32.658, E3 +120759.785}
SPL {X  -157.530, Y  +699.446, Z    +0.000, E1   -24.482, E3 +120762.201}
SPL {X  -159.337, Y  +685.942, Z    +0.000, E1   -14.672, E3 +120763.626}
SPL {X  -159.962, Y  +674.468, Z    +0.000, E1    -4.846, E3 +120764.244}
SPL {X  -159.990, Y  +669.479, Z    +0.000, E1    +0.004, E3 +120764.319}
SPL {X  -159.990, Y  +667.035, Z    +0.000, E1    +4.539, E3 +120764.349}
SPL {X  -159.990, Y  +662.914, Z    +0.000, E1   +13.494, E3 +120764.488}
SPL {X  -159.990, Y  +658.254, Z    +0.000, E1   +24.153, E3 +120764.766}
SPL {X  -159.990, Y  +652.944, Z    +0.000, E1   +35.122, E3 +120765.270}
SPL {X  -159.990, Y  +642.509, Z    +0.000, E1   +50.090, E3 +120766.841}
SPL {X  -159.990, Y  +618.566, Z    +0.000, E1   +64.119, E3 +120773.012}
SPL {X  -159.990, Y  +582.261, Z    +0.000, E1   +69.343, E3 +120786.498}
SPL {X  -159.990, Y  +406.555, Z    +0.000, E1   +71.635, E3 +120882.744}
SPL {X  -159.967, Y  +379.776, Z    +0.000, E1   +71.634, E3 +120901.637}
SPL {X  -158.535, Y  +360.970, Z    +0.000, E1   +71.460, E3 +120916.459}
SPL {X  -156.882, Y  +351.118, Z    +0.000, E1   +71.263, E3 +120925.171}
SPL {X  -155.538, Y  +345.018, Z    +0.000, E1   +71.109, E3 +120930.878}
SPL {X  -155.351, Y  +344.251, Z    +0.000, E1   +70.004, E3 +120941.594}
SPL {X  -150.579, Y  +328.438, Z    +0.000, E1   +70.374, E3 +120949.980}
SPL {X  -146.933, Y  +319.195, Z    +0.000, E1   +70.230, E3 +120957.671}
SPL {X  -143.573, Y  +311.906, Z    +0.000, E1   +69.806, E3 +120965.981}
SPL {X  -140.547, Y  +306.057, Z    +0.000, E1   +69.399, E3 +120972.873}
SPL {X  -137.438, Y  +300.600, Z    +0.000, E1   +68.984, E3 +120979.467}
SPL {X  -133.397, Y  +294.172, Z    +0.000, E1   +68.416, E3 +120987.402}
SPL {X  -128.822, Y  +287.623, Z    +0.000, E1   +67.729, E3 +120995.627}
SPL {X  -124.502, Y  +282.021, Z    +0.000, E1   +67.035, E3 +121002.701}
SPL {X   -85.607, Y  +247.340, Z    +0.000, E1   +53.917, E3 +121146.095}
ENDSPLINE

SPLINE
SPL {X  -134.737, Y  +296.229, Z    +0.000, E1   +47.890, E3 +121288.868}
SPL {X  -154.917, Y  +342.531, Z    +0.000, E1   +31.203, E3 +121307.436}
SPL {X  -159.440, Y  +369.246, Z    +0.000, E1   +13.458, E3 +121311.335}
SPL {X  -159.957, Y  +379.264, Z    +0.000, E1    +4.909, E3 +121311.891}
SPL {X  -159.990, Y  +384.398, Z    +0.000, E1    +0.172, E3 +121311.967}
SPL {X  -159.990, Y  +386.323, Z    +0.000, E1    -3.079, E3 +121311.989}
SPL {X  -159.990, Y  +390.285, Z    +0.000, E1   -11.315, E3 +121312.110}
SPL {X  -159.990, Y  +394.559, Z    +0.000, E1   -20.770, E3 +121312.372}
SPL {X  -159.990, Y  +402.118, Z    +0.000, E1   -35.793, E3 +121313.163}
SPL {X  -159.990, Y  +415.193, Z    +0.000, E1   -52.724, E3 +121315.416}
SPL {X  -159.990, Y  +465.395, Z    +0.000, E1   -68.959, E3 +121330.505}
SPL {X  -159.990, Y  +657.157, Z    +0.000, E1   -72.499, E3 +121426.901}
SPL {X  -159.947, Y  +675.227, Z    +0.000, E1   -72.487, E3 +121439.061}
SPL {X  -159.251, Y  +686.856, Z    +0.000, E1   -72.412, E3 +121447.590}
SPL {X  -157.599, Y  +699.059, Z    +0.000, E1   -72.249, E3 +121457.455}
SPL {X  -155.217, Y  +710.289, Z    +0.000, E1   -71.989, E3 +121467.472}
SPL {X  -152.611, Y  +719.527, Z    +0.000, E1   -71.702, E3 +121476.293}
SPL {X  -149.536, Y  +728.383, Z    +0.000, E1   -71.359, E3 +121485.272}
SPL {X  -146.250, Y  +736.367, Z    +0.000, E1   -70.965, E3 +121493.826}
SPL {X  -143.481, Y  +742.281, Z    +0.000, E1   -70.623, E3 +121500.422}
SPL {X  -140.071, Y  +748.811, Z    +0.000, E1   -70.193, E3 +121507.933}
SPL {X  -136.578, Y  +754.826, Z    +0.000, E1   -69.723, E3 +121515.063}
SPL {X  -133.265, Y  +760.028, Z    +0.000, E1   -69.258, E3 +121521.364}
SPL {X  -130.837, Y  +763.579, Z    +0.000, E1   -68.898, E3 +121525.724}
SPL {X  -127.941, Y  +767.561, Z    +0.000, E1   -68.475, E3 +121530.614}
SPL {X  -123.778, Y  +772.869, Z    +0.000, E1   -67.843, E3 +121537.121}
SPL {X   -84.435, Y  +807.395, Z    +0.000, E1   -55.948, E3 +121649.861}
ENDSPLINE

SPLINE
SPL {X  -119.703, Y  +777.650, Z    +0.000, E1   -51.831, E3 +121813.867}
SPL {X  -145.184, Y  +738.720, Z    +0.000, E1   -43.488, E3 +121840.425}
SPL {X  -154.467, Y  +713.173, Z    +0.000, E1   -32.658, E3 +121848.021}
SPL {X  -157.530, Y  +699.446, Z    +0.000, E1   -24.482, E3 +121850.437}
SPL {X  -159.337, Y  +685.942, Z    +0.000, E1   -14.672, E3 +121851.861}
SPL {X  -159.962, Y  +674.468, Z    +0.000, E1    -4.846, E3 +121852.480}
SPL {X  -159.990, Y  +669.479, Z    +0.000, E1    +0.004, E3 +121852.554}
SPL {X  -159.990, Y  +667.035, Z    +0.000, E1    +4.539, E3 +121852.585}
SPL {X  -159.990, Y  +662.914, Z    +0.000, E1   +13.494, E3 +121852.724}
SPL {X  -159.990, Y  +658.254, Z    +0.000, E1   +24.153, E3 +121853.001}
SPL {X  -159.990, Y  +652.944, Z    +0.000, E1   +35.122, E3 +121853.505}
SPL {X  -159.990, Y  +642.509, Z    +0.000, E1   +50.090, E3 +121855.077}
SPL {X  -159.990, Y  +618.566, Z    +0.000, E1   +64.119, E3 +121861.247}
SPL {X  -159.990, Y  +582.261, Z    +0.000, E1   +69.343, E3 +121874.733}
SPL {X  -159.990, Y  +406.555, Z    +0.000, E1   +71.635, E3 +121970.979}
SPL {X  -159.990, Y  +385.723, Z    +0.000, E1   +71.610, E3 +121985.718}
SPL {X  -159.700, Y  +372.863, Z    +0.000, E1   +71.570, E3 +121995.124}
SPL {X  -158.535, Y  +360.970, Z    +0.000, E1   +71.460, E3 +122004.695}
SPL {X  -156.277, Y  +348.230, Z    +0.000, E1   +71.211, E3 +122016.038}
SPL {X  -155.351, Y  +344.251, Z    +0.000, E1   +70.004, E3 +122029.830}
SPL {X  -150.579, Y  +328.438, Z    +0.000, E1   +70.374, E3 +122038.215}
SPL {X  -146.933, Y  +319.195, Z    +0.000, E1   +70.230, E3 +122045.906}
SPL {X  -143.573, Y  +311.906, Z    +0.000, E1   +69.806, E3 +122054.216}
SPL {X  -139.693, Y  +304.508, Z    +0.000, E1   +69.301, E3 +122062.945}
SPL {X  -135.622, Y  +297.627, Z    +0.000, E1   +68.731, E3 +122071.353}
SPL {X  -132.531, Y  +292.877, Z    +0.000, E1   +68.266, E3 +122077.288}
SPL {X  -128.822, Y  +287.623, Z    +0.000, E1   +67.729, E3 +122083.862}
SPL {X  -124.502, Y  +282.021, Z    +0.000, E1   +67.035, E3 +122090.936}
SPL {X   -85.607, Y  +247.340, Z    +0.000, E1   +53.917, E3 +122234.331}
ENDSPLINE

SPLINE
SPL {X  -134.737, Y  +296.229, Z    +0.000, E1   +47.890, E3 +122377.103}
SPL {X  -154.917, Y  +342.531, Z    +0.000, E1   +31.203, E3 +122395.671}
SPL {X  -159.440, Y  +369.246, Z    +0.000, E1   +13.458, E3 +122399.570}
SPL {X  -159.987, Y  +381.470, Z    +0.000, E1    +2.976, E3 +122400.169}
SPL {X  -159.990, Y  +384.500, Z    +0.000, E1    +0.000, E3 +122400.203}
SPL {X  -159.990, Y  +386.323, Z    +0.000, E1    -3.079, E3 +122400.224}
SPL {X  -159.990, Y  +390.285, Z    +0.000, E1   -11.315, E3 +122400.345}
SPL {X  -159.990, Y  +394.559, Z    +0.000, E1   -20.770, E3 +122400.607}
SPL {X  -159.990, Y  +402.118, Z    +0.000, E1   -35.793, E3 +122401.399}
SPL {X  -159.990, Y  +415.193, Z    +0.000, E1   -52.724, E3 +122403.651}
SPL {X  -159.990, Y  +465.395, Z    +0.000, E1   -68.959, E3 +122418.740}
SPL {X  -159.990, Y  +652.170, Z    +0.000, E1   -72.485, E3 +122511.835}
SPL {X  -159.990, Y  +670.864, Z    +0.000, E1   -72.509, E3 +122524.284}
SPL {X  -159.251, Y  +686.856, Z    +0.000, E1   -72.412, E3 +122535.825}
SPL {X  -157.599, Y  +699.059, Z    +0.000, E1   -72.249, E3 +122545.690}
SPL {X  -155.217, Y  +710.289, Z    +0.000, E1   -71.989, E3 +122555.707}
SPL {X  -152.611, Y  +719.527, Z    +0.000, E1   -71.702, E3 +122564.528}
SPL {X  -149.536, Y  +728.383, Z    +0.000, E1   -71.359, E3 +122573.507}
SPL {X  -146.250, Y  +736.367, Z    +0.000, E1   -70.965, E3 +122582.061}
SPL {X  -143.481, Y  +742.281, Z    +0.000, E1   -70.623, E3 +122588.657}
SPL {X  -140.071, Y  +748.811, Z    +0.000, E1   -70.193, E3 +122596.169}
SPL {X  -136.578, Y  +754.826, Z    +0.000, E1   -69.723, E3 +122603.298}
SPL {X  -133.265, Y  +760.028, Z    +0.000, E1   -69.258, E3 +122609.599}
SPL {X  -129.890, Y  +764.909, Z    +0.000, E1   -68.775, E3 +122615.570}
SPL {X  -125.802, Y  +770.346, Z    +0.000, E1   -68.156, E3 +122622.269}
SPL {X  -122.624, Y  +774.263, Z    +0.000, E1   -67.622, E3 +122627.091}
SPL {X   -84.435, Y  +807.395, Z    +0.000, E1   -55.948, E3 +122738.096}
ENDSPLINE

SPLINE
SPL {X  -119.703, Y  +777.650, Z    +0.000, E1   -51.831, E3 +122902.103}
SPL {X  -145.184, Y  +738.720, Z    +0.000, E1   -43.488, E3 +122928.661}
SPL {X  -156.175, Y  +706.232, Z    +0.000, E1   -28.819, E3 +122937.545}
SPL {X  -159.337, Y  +685.942, Z    +0.000, E1   -14.672, E3 +122940.097}
SPL {X  -159.962, Y  +674.468, Z    +0.000, E1    -4.846, E3 +122940.715}
SPL {X  -159.990, Y  +669.479, Z    +0.000, E1    +0.004, E3 +122940.789}
SPL {X  -159.990, Y  +667.035, Z    +0.000, E1    +4.539, E3 +122940.820}
SPL {X  -159.990, Y  +662.914, Z    +0.000, E1   +13.494, E3 +122940.959}
SPL {X  -159.990, Y  +658.254, Z    +0.000, E1   +24.153, E3 +122941.237}
SPL {X  -159.990, Y  +650.381, Z    +0.000, E1   +39.393, E3 +122942.088}
SPL {X  -159.990, Y  +638.701, Z    +0.000, E1   +53.953, E3 +122943.974}
SPL {X  -159.990, Y  +618.566, Z    +0.000, E1   +64.119, E3 +122949.482}
SPL {X  -159.990, Y  +582.261, Z    +0.000, E1   +69.343, E3 +122962.968}
SPL {X  -159.990, Y  +414.423, Z    +0.000, E1   +71.602, E3 +123053.752}
SPL {X  -159.990, Y  +400.357, Z    +0.000, E1   +71.604, E3 +123063.662}
SPL {X  -159.967, Y  +379.776, Z    +0.000, E1   +71.634, E3 +123078.108}
SPL {X  -158.535, Y  +360.970, Z    +0.000, E1   +71.460, E3 +123092.930}
SPL {X  -156.277, Y  +348.230, Z    +0.000, E1   +71.211, E3 +123104.273}
SPL {X  -155.351, Y  +344.251, Z    +0.000, E1   +70.004, E3 +123118.065}
SPL {X  -150.579, Y  +328.438, Z    +0.000, E1   +70.374, E3 +123126.450}
SPL {X  -146.933, Y  +319.195, Z    +0.000, E1   +70.230, E3 +123134.141}
SPL {X  -143.573, Y  +311.906, Z    +0.000, E1   +69.806, E3 +123142.452}
SPL {X  -139.693, Y  +304.508, Z    +0.000, E1   +69.301, E3 +123151.180}
SPL {X  -135.622, Y  +297.627, Z    +0.000, E1   +68.731, E3 +123159.588}
SPL {X  -131.165, Y  +290.889, Z    +0.000, E1   +68.094, E3 +123167.973}
SPL {X  -126.457, Y  +284.492, Z    +0.000, E1   +67.352, E3 +123176.059}
SPL {X  -123.432, Y  +280.710, Z    +0.000, E1   +66.830, E3 +123180.845}
SPL {X   -85.607, Y  +247.340, Z    +0.000, E1   +53.917, E3 +123322.566}
ENDSPLINE

SPLINE
SPL {X  -134.737, Y  +296.229, Z    +0.000, E1   +47.890, E3 +123465.339}
SPL {X  -154.917, Y  +342.531, Z    +0.000, E1   +31.203, E3 +123483.906}
SPL {X  -159.440, Y  +369.246, Z    +0.000, E1   +13.458, E3 +123487.806}
SPL {X  -159.987, Y  +381.470, Z    +0.000, E1    +2.976, E3 +123488.405}
SPL {X  -159.990, Y  +384.500, Z    +0.000, E1    +0.000, E3 +123488.438}
SPL {X  -159.990, Y  +386.323, Z    +0.000, E1    -3.079, E3 +123488.459}
SPL {X  -159.990, Y  +390.285, Z    +0.000, E1   -11.315, E3 +123488.580}
SPL {X  -159.990, Y  +394.559, Z    +0.000, E1   -20.770, E3 +123488.843}
SPL {X  -159.990, Y  +402.118, Z    +0.000, E1   -35.793, E3 +123489.634}
SPL {X  -159.990, Y  +415.193, Z    +0.000, E1   -52.724, E3 +123491.886}
SPL {X  -159.990, Y  +465.395, Z    +0.000, E1   -68.959, E3 +123506.975}
SPL {X  -159.990, Y  +657.157, Z    +0.000, E1   -72.499, E3 +123603.372}
SPL {X  -159.947, Y  +675.227, Z    +0.000, E1   -72.487, E3 +123615.532}
SPL {X  -159.251, Y  +686.856, Z    +0.000, E1   -72.412, E3 +123624.060}
SPL {X  -157.599, Y  +699.059, Z    +0.000, E1   -72.249, E3 +123633.926}
SPL {X  -155.217, Y  +710.289, Z    +0.000, E1   -71.989, E3 +123643.942}
SPL {X  -152.611, Y  +719.527, Z    +0.000, E1   -71.702, E3 +123652.763}
SPL {X  -149.536, Y  +728.383, Z    +0.000, E1   -71.359, E3 +123661.743}
SPL {X  -146.250, Y  +736.367, Z    +0.000, E1   -70.965, E3 +123670.297}
SPL {X  -143.481, Y  +742.281, Z    +0.000, E1   -70.623, E3 +123676.892}
SPL {X  -140.071, Y  +748.811, Z    +0.000, E1   -70.193, E3 +123684.404}
SPL {X  -136.578, Y  +754.826, Z    +0.000, E1   -69.723, E3 +123691.533}
SPL {X  -132.176, Y  +761.646, Z    +0.000, E1   -69.128, E3 +123699.777}
SPL {X  -127.941, Y  +767.561, Z    +0.000, E1   -68.475, E3 +123707.085}
SPL {X  -123.778, Y  +772.869, Z    +0.000, E1   -67.843, E3 +123713.592}
SPL {X   -84.435, Y  +807.395, Z    +0.000, E1   -55.948, E3 +123826.331}
ENDSPLINE

SPLINE
SPL {X  -119.703, Y  +777.650, Z    +0.000, E1   -51.831, E3 +123990.338}
SPL {X  -145.184, Y  +738.720, Z    +0.000, E1   -43.488, E3 +124016.896}
SPL {X  -154.467, Y  +713.173, Z    +0.000, E1   -32.658, E3 +124024.491}
SPL {X  -157.530, Y  +699.446, Z    +0.000, E1   -24.482, E3 +124026.907}
SPL {X  -159.337, Y  +685.942, Z    +0.000, E1   -14.672, E3 +124028.332}
SPL {X  -159.900, Y  +676.871, Z    +0.000, E1    -6.955, E3 +124028.880}
SPL {X  -159.990, Y  +669.634, Z    +0.000, E1    -0.285, E3 +124029.023}
SPL {X  -159.990, Y  +667.035, Z    +0.000, E1    +4.539, E3 +124029.055}
SPL {X  -159.990, Y  +662.914, Z    +0.000, E1   +13.494, E3 +124029.194}
SPL {X  -159.990, Y  +658.254, Z    +0.000, E1   +24.153, E3 +124029.472}
SPL {X  -159.990, Y  +650.381, Z    +0.000, E1   +39.393, E3 +124030.324}
SPL {X  -159.990, Y  +638.701, Z    +0.000, E1   +53.953, E3 +124032.210}
SPL {X  -159.990, Y  +618.566, Z    +0.000, E1   +64.119, E3 +124037.718}
SPL {X  -159.990, Y  +582.261, Z    +0.000, E1   +69.343, E3 +124051.204}
SPL {X  -159.990, Y  +406.555, Z    +0.000, E1   +71.635, E3 +124147.450}
SPL {X  -159.990, Y  +385.723, Z    +0.000, E1   +71.610, E3 +124162.188}
SPL {X  -159.404, Y  +368.814, Z    +0.000, E1   +71.556, E3 +124174.718}
SPL {X  -158.061, Y  +357.731, Z    +0.000, E1   +71.393, E3 +124183.986}
SPL {X  -156.277, Y  +348.230, Z    +0.000, E1   +71.211, E3 +124192.508}
SPL {X  -155.351, Y  +344.251, Z    +0.000, E1   +70.004, E3 +124206.300}
SPL {X  -150.579, Y  +328.438, Z    +0.000, E1   +70.374, E3 +124214.686}
SPL {X  -146.933, Y  +319.195, Z    +0.000, E1   +70.230, E3 +124222.377}
SPL {X  -143.573, Y  +311.906, Z    +0.000, E1   +69.806, E3 +124230.687}
SPL {X  -140.547, Y  +306.057, Z    +0.000, E1   +69.399, E3 +124237.579}
SPL {X  -137.438, Y  +300.600, Z    +0.000, E1   +68.984, E3 +124244.173}
SPL {X  -133.397, Y  +294.172, Z    +0.000, E1   +68.416, E3 +124252.108}
SPL {X  -128.822, Y  +287.623, Z    +0.000, E1   +67.729, E3 +124260.333}
SPL {X  -124.502, Y  +282.021, Z    +0.000, E1   +67.035, E3 +124267.407}
SPL {X   -85.607, Y  +247.340, Z    +0.000, E1   +53.917, E3 +124410.801}
ENDSPLINE

SPLINE
SPL {X  -134.737, Y  +296.229, Z    +0.000, E1   +47.890, E3 +124553.574}
SPL {X  -154.917, Y  +342.531, Z    +0.000, E1   +31.203, E3 +124572.142}
SPL {X  -159.440, Y  +369.246, Z    +0.000, E1   +13.458, E3 +124576.041}
SPL {X  -159.987, Y  +381.470, Z    +0.000, E1    +2.976, E3 +124576.640}
SPL {X  -159.990, Y  +384.500, Z    +0.000, E1    +0.000, E3 +124576.673}
SPL {X  -159.990, Y  +386.323, Z    +0.000, E1    -3.079, E3 +124576.695}
SPL {X  -159.990, Y  +390.285, Z    +0.000, E1   -11.315, E3 +124576.816}
SPL {X  -159.990, Y  +394.559, Z    +0.000, E1   -20.770, E3 +124577.078}
SPL {X  -159.990, Y  +399.334, Z    +0.000, E1   -30.876, E3 +124577.517}
SPL {X  -159.990, Y  +405.006, Z    +0.000, E1   -40.810, E3 +124578.235}
SPL {X  -159.990, Y  +415.193, Z    +0.000, E1   -52.724, E3 +124580.122}
SPL {X  -159.990, Y  +465.395, Z    +0.000, E1   -68.959, E3 +124595.210}
SPL {X  -159.990, Y  +657.157, Z    +0.000, E1   -72.499, E3 +124691.607}
SPL {X  -159.693, Y  +681.249, Z    +0.000, E1   -72.488, E3 +124708.001}
SPL {X  -157.599, Y  +699.059, Z    +0.000, E1   -72.249, E3 +124722.161}
SPL {X  -155.217, Y  +710.289, Z    +0.000, E1   -71.989, E3 +124732.177}
SPL {X  -152.611, Y  +719.527, Z    +0.000, E1   -71.702, E3 +124740.999}
SPL {X  -149.536, Y  +728.383, Z    +0.000, E1   -71.359, E3 +124749.978}
SPL {X  -146.250, Y  +736.367, Z    +0.000, E1   -70.965, E3 +124758.532}
SPL {X  -143.481, Y  +742.281, Z    +0.000, E1   -70.623, E3 +124765.128}
SPL {X  -140.071, Y  +748.811, Z    +0.000, E1   -70.193, E3 +124772.639}
SPL {X  -136.578, Y  +754.826, Z    +0.000, E1   -69.723, E3 +124779.769}
SPL {X  -133.265, Y  +760.028, Z    +0.000, E1   -69.258, E3 +124786.070}
SPL {X  -130.837, Y  +763.579, Z    +0.000, E1   -68.898, E3 +124790.430}
SPL {X  -127.941, Y  +767.561, Z    +0.000, E1   -68.475, E3 +124795.320}
SPL {X  -123.778, Y  +772.869, Z    +0.000, E1   -67.843, E3 +124801.827}
SPL {X   -84.435, Y  +807.395, Z    +0.000, E1   -55.948, E3 +124914.566}
ENDSPLINE

SPLINE
SPL {X  -119.703, Y  +777.650, Z    +0.000, E1   -51.831, E3 +125078.573}
SPL {X  -145.184, Y  +738.720, Z    +0.000, E1   -43.488, E3 +125105.131}
SPL {X  -156.175, Y  +706.232, Z    +0.000, E1   -28.819, E3 +125114.016}
SPL {X  -159.337, Y  +685.942, Z    +0.000, E1   -14.672, E3 +125116.567}
SPL {X  -159.962, Y  +674.468, Z    +0.000, E1    -4.846, E3 +125117.186}
SPL {X  -159.990, Y  +669.479, Z    +0.000, E1    +0.004, E3 +125117.260}
SPL {X  -159.990, Y  +667.035, Z    +0.000, E1    +4.539, E3 +125117.291}
SPL {X  -159.990, Y  +662.914, Z    +0.000, E1   +13.494, E3 +125117.430}
SPL {X  -159.990, Y  +658.254, Z    +0.000, E1   +24.153, E3 +125117.707}
SPL {X  -159.990, Y  +652.944, Z    +0.000, E1   +35.122, E3 +125118.211}
SPL {X  -159.990, Y  +646.557, Z    +0.000, E1   +45.390, E3 +125119.078}
SPL {X  -159.990, Y  +638.701, Z    +0.000, E1   +53.953, E3 +125120.445}
SPL {X  -159.990, Y  +618.566, Z    +0.000, E1   +64.119, E3 +125125.953}
SPL {X  -159.990, Y  +582.261, Z    +0.000, E1   +69.343, E3 +125139.439}
SPL {X  -159.990, Y  +426.570, Z    +0.000, E1   +71.599, E3 +125221.702}
SPL {X  -159.990, Y  +405.946, Z    +0.000, E1   +71.630, E3 +125236.132}
SPL {X  -159.990, Y  +385.723, Z    +0.000, E1   +71.610, E3 +125250.424}
SPL {X  -159.404, Y  +368.814, Z    +0.000, E1   +71.556, E3 +125262.953}
SPL {X  -158.061, Y  +357.731, Z    +0.000, E1   +71.393, E3 +125272.221}
SPL {X  -156.277, Y  +348.230, Z    +0.000, E1   +71.211, E3 +125280.744}
SPL {X  -155.351, Y  +344.251, Z    +0.000, E1   +70.004, E3 +125294.536}
SPL {X  -150.579, Y  +328.438, Z    +0.000, E1   +70.374, E3 +125302.921}
SPL {X  -146.933, Y  +319.195, Z    +0.000, E1   +70.230, E3 +125310.612}
SPL {X  -143.573, Y  +311.906, Z    +0.000, E1   +69.806, E3 +125318.922}
SPL {X  -140.547, Y  +306.057, Z    +0.000, E1   +69.399, E3 +125325.814}
SPL {X  -136.400, Y  +298.883, Z    +0.000, E1   +68.867, E3 +125334.470}
SPL {X  -131.165, Y  +290.889, Z    +0.000, E1   +68.094, E3 +125344.444}
SPL {X  -126.457, Y  +284.492, Z    +0.000, E1   +67.352, E3 +125352.529}
SPL {X  -123.432, Y  +280.710, Z    +0.000, E1   +66.830, E3 +125357.315}
SPL {X   -85.607, Y  +247.340, Z    +0.000, E1   +53.917, E3 +125499.036}
ENDSPLINE

SPLINE
SPL {X  -119.557, Y  +276.184, Z    +0.000, E1   +51.032, E3 +125622.573}
SPL {X  -138.294, Y  +302.054, Z    +0.000, E1   +46.576, E3 +125645.895}
SPL {X  -153.211, Y  +336.421, Z    +0.000, E1   +34.262, E3 +125659.017}
SPL {X  -158.240, Y  +358.900, Z    +0.000, E1   +21.089, E3 +125663.223}
SPL {X  -159.674, Y  +372.451, Z    +0.000, E1   +10.778, E3 +125664.518}
SPL {X  -159.987, Y  +381.470, Z    +0.000, E1    +2.976, E3 +125664.875}
SPL {X  -159.990, Y  +384.761, Z    +0.000, E1    -0.257, E3 +125664.910}
SPL {X  -159.990, Y  +389.248, Z    +0.000, E1    -8.879, E3 +125665.014}
SPL {X  -159.990, Y  +394.559, Z    +0.000, E1   -20.770, E3 +125665.313}
SPL {X  -159.990, Y  +402.118, Z    +0.000, E1   -35.793, E3 +125666.105}
SPL {X  -159.990, Y  +415.193, Z    +0.000, E1   -52.724, E3 +125668.357}
SPL {X  -159.990, Y  +465.395, Z    +0.000, E1   -68.959, E3 +125683.446}
SPL {X  -159.990, Y  +657.157, Z    +0.000, E1   -72.499, E3 +125779.842}
SPL {X  -159.947, Y  +675.227, Z    +0.000, E1   -72.487, E3 +125792.003}
SPL {X  -159.251, Y  +686.856, Z    +0.000, E1   -72.412, E3 +125800.531}
SPL {X  -157.599, Y  +699.059, Z    +0.000, E1   -72.249, E3 +125810.396}
SPL {X  -155.217, Y  +710.289, Z    +0.000, E1   -71.989, E3 +125820.413}
SPL {X  -152.611, Y  +719.527, Z    +0.000, E1   -71.702, E3 +125829.234}
SPL {X  -149.536, Y  +728.383, Z    +0.000, E1   -71.359, E3 +125838.213}
SPL {X  -146.250, Y  +736.367, Z    +0.000, E1   -70.965, E3 +125846.767}
SPL {X  -143.481, Y  +742.281, Z    +0.000, E1   -70.623, E3 +125853.363}
SPL {X  -140.071, Y  +748.811, Z    +0.000, E1   -70.193, E3 +125860.875}
SPL {X  -136.578, Y  +754.826, Z    +0.000, E1   -69.723, E3 +125868.004}
SPL {X  -133.265, Y  +760.028, Z    +0.000, E1   -69.258, E3 +125874.305}
SPL {X  -129.890, Y  +764.909, Z    +0.000, E1   -68.775, E3 +125880.276}
SPL {X  -125.802, Y  +770.346, Z    +0.000, E1   -68.156, E3 +125886.975}
SPL {X  -122.624, Y  +774.263, Z    +0.000, E1   -67.622, E3 +125891.797}
SPL {X   -84.435, Y  +807.395, Z    +0.000, E1   -55.948, E3 +126002.802}
ENDSPLINE

SPLINE
SPL {X  -119.703, Y  +777.650, Z    +0.000, E1   -51.831, E3 +126166.808}
SPL {X  -145.184, Y  +738.720, Z    +0.000, E1   -43.488, E3 +126193.366}
SPL {X  -154.467, Y  +713.173, Z    +0.000, E1   -32.658, E3 +126200.962}
SPL {X  -157.530, Y  +699.446, Z    +0.000, E1   -24.482, E3 +126203.378}
SPL {X  -159.337, Y  +685.942, Z    +0.000, E1   -14.672, E3 +126204.802}
SPL {X  -159.962, Y  +674.468, Z    +0.000, E1    -4.846, E3 +126205.421}
SPL {X  -159.990, Y  +669.479, Z    +0.000, E1    +0.004, E3 +126205.495}
SPL {X  -159.990, Y  +667.035, Z    +0.000, E1    +4.539, E3 +126205.526}
SPL {X  -159.990, Y  +662.914, Z    +0.000, E1   +13.494, E3 +126205.665}
SPL {X  -159.990, Y  +658.254, Z    +0.000, E1   +24.153, E3 +126205.943}
SPL {X  -159.990, Y  +652.944, Z    +0.000, E1   +35.122, E3 +126206.446}
SPL {X  -159.990, Y  +642.509, Z    +0.000, E1   +50.090, E3 +126208.018}
SPL {X  -159.990, Y  +618.566, Z    +0.000, E1   +64.119, E3 +126214.188}
SPL {X  -159.990, Y  +582.261, Z    +0.000, E1   +69.343, E3 +126227.674}
SPL {X  -159.990, Y  +406.555, Z    +0.000, E1   +71.635, E3 +126323.921}
SPL {X  -159.967, Y  +379.776, Z    +0.000, E1   +71.634, E3 +126342.814}
SPL {X  -158.535, Y  +360.970, Z    +0.000, E1   +71.460, E3 +126357.636}
SPL {X  -156.882, Y  +351.118, Z    +0.000, E1   +71.263, E3 +126366.348}
SPL {X  -155.538, Y  +345.018, Z    +0.000, E1   +71.109, E3 +126372.054}
SPL {X  -155.351, Y  +344.251, Z    +0.000, E1   +70.004, E3 +126382.771}
SPL {X  -150.579, Y  +328.438, Z    +0.000, E1   +70.374, E3 +126391.156}
SPL {X  -146.933, Y  +319.195, Z    +0.000, E1   +70.230, E3 +126398.847}
SPL {X  -143.573, Y  +311.906, Z    +0.000, E1   +69.806, E3 +126407.158}
SPL {X  -140.547, Y  +306.057, Z    +0.000, E1   +69.399, E3 +126414.049}
SPL {X  -137.438, Y  +300.600, Z    +0.000, E1   +68.984, E3 +126420.644}
SPL {X  -133.397, Y  +294.172, Z    +0.000, E1   +68.416, E3 +126428.579}
SPL {X  -128.822, Y  +287.623, Z    +0.000, E1   +67.729, E3 +126436.803}
SPL {X  -124.502, Y  +282.021, Z    +0.000, E1   +67.035, E3 +126443.877}
SPL {X   -85.607, Y  +247.340, Z    +0.000, E1   +53.917, E3 +126587.272}
ENDSPLINE

SPLINE
SPL {X  -134.737, Y  +296.229, Z    +0.000, E1   +47.890, E3 +126730.045}
SPL {X  -154.917, Y  +342.531, Z    +0.000, E1   +31.203, E3 +126748.612}
SPL {X  -159.440, Y  +369.246, Z    +0.000, E1   +13.458, E3 +126752.511}
SPL {X  -159.957, Y  +379.264, Z    +0.000, E1    +4.909, E3 +126753.068}
SPL {X  -159.990, Y  +384.398, Z    +0.000, E1    +0.172, E3 +126753.143}
SPL {X  -159.990, Y  +386.323, Z    +0.000, E1    -3.079, E3 +126753.165}
SPL {X  -159.990, Y  +390.285, Z    +0.000, E1   -11.315, E3 +126753.286}
SPL {X  -159.990, Y  +394.559, Z    +0.000, E1   -20.770, E3 +126753.548}
SPL {X  -159.990, Y  +402.118, Z    +0.000, E1   -35.793, E3 +126754.340}
SPL {X  -159.990, Y  +415.193, Z    +0.000, E1   -52.724, E3 +126756.592}
SPL {X  -159.990, Y  +465.395, Z    +0.000, E1   -68.959, E3 +126771.681}
SPL {X  -159.990, Y  +657.157, Z    +0.000, E1   -72.499, E3 +126868.078}
SPL {X  -159.693, Y  +681.249, Z    +0.000, E1   -72.488, E3 +126884.472}
SPL {X  -157.599, Y  +699.059, Z    +0.000, E1   -72.249, E3 +126898.631}
SPL {X  -155.217, Y  +710.289, Z    +0.000, E1   -71.989, E3 +126908.648}
SPL {X  -152.611, Y  +719.527, Z    +0.000, E1   -71.702, E3 +126917.469}
SPL {X  -149.536, Y  +728.383, Z    +0.000, E1   -71.359, E3 +126926.449}
SPL {X  -146.250, Y  +736.367, Z    +0.000, E1   -70.965, E3 +126935.003}
SPL {X  -143.481, Y  +742.281, Z    +0.000, E1   -70.623, E3 +126941.598}
SPL {X  -140.071, Y  +748.811, Z    +0.000, E1   -70.193, E3 +126949.110}
SPL {X  -136.578, Y  +754.826, Z    +0.000, E1   -69.723, E3 +126956.239}
SPL {X  -132.176, Y  +761.646, Z    +0.000, E1   -69.128, E3 +126964.483}
SPL {X  -127.941, Y  +767.561, Z    +0.000, E1   -68.475, E3 +126971.791}
SPL {X  -123.778, Y  +772.869, Z    +0.000, E1   -67.843, E3 +126978.298}
SPL {X   -84.435, Y  +807.395, Z    +0.000, E1   -55.948, E3 +127091.037}
ENDSPLINE

SPLINE
SPL {X  -119.703, Y  +777.650, Z    +0.000, E1   -51.831, E3 +127255.044}
SPL {X  -145.184, Y  +738.720, Z    +0.000, E1   -43.488, E3 +127281.602}
SPL {X  -156.175, Y  +706.232, Z    +0.000, E1   -28.819, E3 +127290.487}
SPL {X  -159.337, Y  +685.942, Z    +0.000, E1   -14.672, E3 +127293.038}
SPL {X  -159.900, Y  +676.871, Z    +0.000, E1    -6.955, E3 +127293.586}
SPL {X  -159.990, Y  +669.634, Z    +0.000, E1    -0.285, E3 +127293.729}
SPL {X  -159.990, Y  +667.035, Z    +0.000, E1    +4.539, E3 +127293.761}
SPL {X  -159.990, Y  +662.914, Z    +0.000, E1   +13.494, E3 +127293.900}
SPL {X  -159.990, Y  +658.254, Z    +0.000, E1   +24.153, E3 +127294.178}
SPL {X  -159.990, Y  +650.381, Z    +0.000, E1   +39.393, E3 +127295.029}
SPL {X  -159.990, Y  +638.701, Z    +0.000, E1   +53.953, E3 +127296.915}
SPL {X  -159.990, Y  +618.566, Z    +0.000, E1   +64.119, E3 +127302.424}
SPL {X  -159.990, Y  +582.261, Z    +0.000, E1   +69.343, E3 +127315.909}
SPL {X  -159.990, Y  +406.555, Z    +0.000, E1   +71.635, E3 +127412.156}
SPL {X  -159.967, Y  +379.776, Z    +0.000, E1   +71.634, E3 +127431.049}
SPL {X  -158.535, Y  +360.970, Z    +0.000, E1   +71.460, E3 +127445.871}
SPL {X  -156.277, Y  +348.230, Z    +0.000, E1   +71.211, E3 +127457.214}
SPL {X  -155.351, Y  +344.251, Z    +0.000, E1   +70.004, E3 +127471.006}
SPL {X  -150.579, Y  +328.438, Z    +0.000, E1   +70.374, E3 +127479.392}
SPL {X  -146.933, Y  +319.195, Z    +0.000, E1   +70.230, E3 +127487.082}
SPL {X  -143.573, Y  +311.906, Z    +0.000, E1   +69.806, E3 +127495.393}
SPL {X  -139.693, Y  +304.508, Z    +0.000, E1   +69.301, E3 +127504.121}
SPL {X  -135.622, Y  +297.627, Z    +0.000, E1   +68.731, E3 +127512.529}
SPL {X  -131.165, Y  +290.889, Z    +0.000, E1   +68.094, E3 +127520.914}
SPL {X  -126.457, Y  +284.492, Z    +0.000, E1   +67.352, E3 +127529.000}
SPL {X  -123.432, Y  +280.710, Z    +0.000, E1   +66.830, E3 +127533.786}
SPL {X   -85.607, Y  +247.340, Z    +0.000, E1   +53.917, E3 +127675.507}
ENDSPLINE

SPLINE
SPL {X  -134.737, Y  +296.229, Z    +0.000, E1   +47.890, E3 +127818.280}
SPL {X  -154.917, Y  +342.531, Z    +0.000, E1   +31.203, E3 +127836.848}
SPL {X  -159.440, Y  +369.246, Z    +0.000, E1   +13.458, E3 +127840.747}
SPL {X  -159.987, Y  +381.470, Z    +0.000, E1    +2.976, E3 +127841.346}
SPL {X  -159.990, Y  +384.500, Z    +0.000, E1    +0.000, E3 +127841.379}
SPL {X  -159.990, Y  +386.323, Z    +0.000, E1    -3.079, E3 +127841.400}
SPL {X  -159.990, Y  +390.285, Z    +0.000, E1   -11.315, E3 +127841.522}
SPL {X  -159.990, Y  +394.559, Z    +0.000, E1   -20.770, E3 +127841.784}
SPL {X  -159.990, Y  +399.334, Z    +0.000, E1   -30.876, E3 +127842.223}
SPL {X  -159.990, Y  +405.006, Z    +0.000, E1   -40.810, E3 +127842.941}
SPL {X  -159.990, Y  +415.193, Z    +0.000, E1   -52.724, E3 +127844.828}
SPL {X  -159.990, Y  +465.395, Z    +0.000, E1   -68.959, E3 +127859.916}
SPL {X  -159.990, Y  +657.157, Z    +0.000, E1   -72.499, E3 +127956.313}
SPL {X  -159.693, Y  +681.249, Z    +0.000, E1   -72.488, E3 +127972.707}
SPL {X  -157.599, Y  +699.059, Z    +0.000, E1   -72.249, E3 +127986.867}
SPL {X  -155.217, Y  +710.289, Z    +0.000, E1   -71.989, E3 +127996.883}
SPL {X  -152.611, Y  +719.527, Z    +0.000, E1   -71.702, E3 +128005.705}
SPL {X  -149.536, Y  +728.383, Z    +0.000, E1   -71.359, E3 +128014.684}
SPL {X  -146.250, Y  +736.367, Z    +0.000, E1   -70.965, E3 +128023.238}
SPL {X  -143.481, Y  +742.281, Z    +0.000, E1   -70.623, E3 +128029.833}
SPL {X  -140.071, Y  +748.811, Z    +0.000, E1   -70.193, E3 +128037.345}
SPL {X  -136.578, Y  +754.826, Z    +0.000, E1   -69.723, E3 +128044.475}
SPL {X  -133.265, Y  +760.028, Z    +0.000, E1   -69.258, E3 +128050.775}
SPL {X  -130.837, Y  +763.579, Z    +0.000, E1   -68.898, E3 +128055.136}
SPL {X  -127.941, Y  +767.561, Z    +0.000, E1   -68.475, E3 +128060.026}
SPL {X  -123.778, Y  +772.869, Z    +0.000, E1   -67.843, E3 +128066.533}
SPL {X   -84.435, Y  +807.395, Z    +0.000, E1   -55.948, E3 +128179.272}
ENDSPLINE

SPLINE
SPL {X  -119.703, Y  +777.650, Z    +0.000, E1   -51.831, E3 +128343.279}
SPL {X  -145.184, Y  +738.720, Z    +0.000, E1   -43.488, E3 +128369.837}
SPL {X  -156.175, Y  +706.232, Z    +0.000, E1   -28.819, E3 +128378.722}
SPL {X  -159.337, Y  +685.942, Z    +0.000, E1   -14.672, E3 +128381.273}
SPL {X  -159.962, Y  +674.468, Z    +0.000, E1    -4.846, E3 +128381.892}
SPL {X  -159.990, Y  +669.479, Z    +0.000, E1    +0.004, E3 +128381.966}
SPL {X  -159.990, Y  +667.035, Z    +0.000, E1    +4.539, E3 +128381.997}
SPL {X  -159.990, Y  +662.914, Z    +0.000, E1   +13.494, E3 +128382.135}
SPL {X  -159.990, Y  +658.254, Z    +0.000, E1   +24.153, E3 +128382.413}
SPL {X  -159.990, Y  +652.944, Z    +0.000, E1   +35.122, E3 +128382.917}
SPL {X  -159.990, Y  +646.557, Z    +0.000, E1   +45.390, E3 +128383.784}
SPL {X  -159.990, Y  +638.701, Z    +0.000, E1   +53.953, E3 +128385.151}
SPL {X  -159.990, Y  +618.566, Z    +0.000, E1   +64.119, E3 +128390.659}
SPL {X  -159.990, Y  +582.261, Z    +0.000, E1   +69.343, E3 +128404.145}
SPL {X  -159.990, Y  +426.570, Z    +0.000, E1   +71.599, E3 +128486.408}
SPL {X  -159.990, Y  +405.946, Z    +0.000, E1   +71.630, E3 +128500.838}
SPL {X  -159.990, Y  +385.723, Z    +0.000, E1   +71.610, E3 +128515.129}
SPL {X  -159.404, Y  +368.814, Z    +0.000, E1   +71.556, E3 +128527.659}
SPL {X  -158.061, Y  +357.731, Z    +0.000, E1   +71.393, E3 +128536.927}
SPL {X  -156.277, Y  +348.230, Z    +0.000, E1   +71.211, E3 +128545.450}
SPL {X  -155.351, Y  +344.251, Z    +0.000, E1   +70.004, E3 +128559.241}
SPL {X  -150.579, Y  +328.438, Z    +0.000, E1   +70.374, E3 +128567.627}
SPL {X  -146.933, Y  +319.195, Z    +0.000, E1   +70.230, E3 +128575.318}
SPL {X  -143.573, Y  +311.906, Z    +0.000, E1   +69.806, E3 +128583.628}
SPL {X  -140.547, Y  +306.057, Z    +0.000, E1   +69.399, E3 +128590.520}
SPL {X  -136.400, Y  +298.883, Z    +0.000, E1   +68.867, E3 +128599.176}
SPL {X  -131.165, Y  +290.889, Z    +0.000, E1   +68.094, E3 +128609.150}
SPL {X  -126.457, Y  +284.492, Z    +0.000, E1   +67.352, E3 +128617.235}
SPL {X  -123.432, Y  +280.710, Z    +0.000, E1   +66.830, E3 +128622.021}
SPL {X   -85.607, Y  +247.340, Z    +0.000, E1   +53.917, E3 +128763.742}
ENDSPLINE

SPLINE
SPL {X  -119.557, Y  +276.184, Z    +0.000, E1   +51.032, E3 +128887.279}
SPL {X  -138.294, Y  +302.054, Z    +0.000, E1   +46.576, E3 +128910.601}
SPL {X  -153.211, Y  +336.421, Z    +0.000, E1   +34.262, E3 +128923.723}
SPL {X  -158.240, Y  +358.900, Z    +0.000, E1   +21.089, E3 +128927.928}
SPL {X  -159.674, Y  +372.451, Z    +0.000, E1   +10.778, E3 +128929.224}
SPL {X  -159.987, Y  +381.470, Z    +0.000, E1    +2.976, E3 +128929.581}
SPL {X  -159.990, Y  +384.761, Z    +0.000, E1    -0.257, E3 +128929.616}
SPL {X  -159.990, Y  +389.248, Z    +0.000, E1    -8.879, E3 +128929.720}
SPL {X  -159.990, Y  +394.559, Z    +0.000, E1   -20.770, E3 +128930.019}
SPL {X  -159.990, Y  +402.118, Z    +0.000, E1   -35.793, E3 +128930.810}
SPL {X  -159.990, Y  +415.193, Z    +0.000, E1   -52.724, E3 +128933.063}
SPL {X  -159.990, Y  +465.395, Z    +0.000, E1   -68.959, E3 +128948.152}
SPL {X  -159.990, Y  +657.157, Z    +0.000, E1   -72.499, E3 +129044.548}
SPL {X  -159.693, Y  +681.249, Z    +0.000, E1   -72.488, E3 +129060.942}
SPL {X  -157.599, Y  +699.059, Z    +0.000, E1   -72.249, E3 +129075.102}
SPL {X  -155.217, Y  +710.289, Z    +0.000, E1   -71.989, E3 +129085.119}
SPL {X  -152.611, Y  +719.527, Z    +0.000, E1   -71.702, E3 +129093.940}
SPL {X  -149.536, Y  +728.383, Z    +0.000, E1   -71.359, E3 +129102.919}
SPL {X  -146.250, Y  +736.367, Z    +0.000, E1   -70.965, E3 +129111.473}
SPL {X  -143.481, Y  +742.281, Z    +0.000, E1   -70.623, E3 +129118.069}
SPL {X  -140.071, Y  +748.811, Z    +0.000, E1   -70.193, E3 +129125.580}
SPL {X  -136.578, Y  +754.826, Z    +0.000, E1   -69.723, E3 +129132.710}
SPL {X  -133.265, Y  +760.028, Z    +0.000, E1   -69.258, E3 +129139.011}
SPL {X  -129.890, Y  +764.909, Z    +0.000, E1   -68.775, E3 +129144.981}
SPL {X  -125.802, Y  +770.346, Z    +0.000, E1   -68.156, E3 +129151.681}
SPL {X  -122.624, Y  +774.263, Z    +0.000, E1   -67.622, E3 +129156.503}
SPL {X   -84.435, Y  +807.395, Z    +0.000, E1   -55.948, E3 +129267.508}
ENDSPLINE

SPLINE
SPL {X  -119.703, Y  +777.650, Z    +0.000, E1   -51.831, E3 +129431.514}
SPL {X  -145.184, Y  +738.720, Z    +0.000, E1   -43.488, E3 +129458.072}
SPL {X  -156.175, Y  +706.232, Z    +0.000, E1   -28.819, E3 +129466.957}
SPL {X  -159.337, Y  +685.942, Z    +0.000, E1   -14.672, E3 +129469.508}
SPL {X  -159.900, Y  +676.871, Z    +0.000, E1    -6.955, E3 +129470.056}
SPL {X  -159.990, Y  +669.634, Z    +0.000, E1    -0.285, E3 +129470.200}
SPL {X  -159.990, Y  +667.035, Z    +0.000, E1    +4.539, E3 +129470.232}
SPL {X  -159.990, Y  +662.914, Z    +0.000, E1   +13.494, E3 +129470.371}
SPL {X  -159.990, Y  +658.254, Z    +0.000, E1   +24.153, E3 +129470.648}
SPL {X  -159.990, Y  +652.944, Z    +0.000, E1   +35.122, E3 +129471.152}
SPL {X  -159.990, Y  +642.509, Z    +0.000, E1   +50.090, E3 +129472.724}
SPL {X  -159.990, Y  +618.566, Z    +0.000, E1   +64.119, E3 +129478.894}
SPL {X  -159.990, Y  +582.261, Z    +0.000, E1   +69.343, E3 +129492.380}
SPL {X  -159.990, Y  +406.555, Z    +0.000, E1   +71.635, E3 +129588.627}
SPL {X  -159.967, Y  +379.776, Z    +0.000, E1   +71.634, E3 +129607.520}
SPL {X  -158.535, Y  +360.970, Z    +0.000, E1   +71.460, E3 +129622.342}
SPL {X  -156.882, Y  +351.118, Z    +0.000, E1   +71.263, E3 +129631.053}
SPL {X  -155.538, Y  +345.018, Z    +0.000, E1   +71.109, E3 +129636.760}
SPL {X  -155.351, Y  +344.251, Z    +0.000, E1   +70.004, E3 +129647.477}
SPL {X  -150.579, Y  +328.438, Z    +0.000, E1   +70.374, E3 +129655.862}
SPL {X  -146.933, Y  +319.195, Z    +0.000, E1   +70.230, E3 +129663.553}
SPL {X  -143.573, Y  +311.906, Z    +0.000, E1   +69.806, E3 +129671.863}
SPL {X  -140.547, Y  +306.057, Z    +0.000, E1   +69.399, E3 +129678.755}
SPL {X  -136.400, Y  +298.883, Z    +0.000, E1   +68.867, E3 +129687.411}
SPL {X  -131.165, Y  +290.889, Z    +0.000, E1   +68.094, E3 +129697.385}
SPL {X  -126.457, Y  +284.492, Z    +0.000, E1   +67.352, E3 +129705.470}
SPL {X  -123.432, Y  +280.710, Z    +0.000, E1   +66.830, E3 +129710.256}
SPL {X   -85.607, Y  +247.340, Z    +0.000, E1   +53.917, E3 +129851.978}
ENDSPLINE

SPLINE
SPL {X  -119.557, Y  +276.184, Z    +0.000, E1   +51.032, E3 +129975.514}
SPL {X  -138.294, Y  +302.054, Z    +0.000, E1   +46.576, E3 +129998.836}
SPL {X  -153.211, Y  +336.421, Z    +0.000, E1   +34.262, E3 +130011.958}
SPL {X  -158.240, Y  +358.900, Z    +0.000, E1   +21.089, E3 +130016.164}
SPL {X  -159.854, Y  +375.896, Z    +0.000, E1    +7.981, E3 +130017.630}
SPL {X  -159.990, Y  +384.398, Z    +0.000, E1    +0.172, E3 +130017.849}
SPL {X  -159.990, Y  +386.323, Z    +0.000, E1    -3.079, E3 +130017.871}
SPL {X  -159.990, Y  +390.285, Z    +0.000, E1   -11.315, E3 +130017.992}
SPL {X  -159.990, Y  +394.559, Z    +0.000, E1   -20.770, E3 +130018.254}
SPL {X  -159.990, Y  +399.334, Z    +0.000, E1   -30.876, E3 +130018.693}
SPL {X  -159.990, Y  +405.006, Z    +0.000, E1   -40.810, E3 +130019.411}
SPL {X  -159.990, Y  +415.193, Z    +0.000, E1   -52.724, E3 +130021.298}
SPL {X  -159.990, Y  +465.395, Z    +0.000, E1   -68.959, E3 +130036.387}
SPL {X  -159.990, Y  +657.157, Z    +0.000, E1   -72.499, E3 +130132.784}
SPL {X  -159.693, Y  +681.249, Z    +0.000, E1   -72.488, E3 +130149.178}
SPL {X  -157.599, Y  +699.059, Z    +0.000, E1   -72.249, E3 +130163.337}
SPL {X  -155.217, Y  +710.289, Z    +0.000, E1   -71.989, E3 +130173.354}
SPL {X  -152.611, Y  +719.527, Z    +0.000, E1   -71.702, E3 +130182.175}
SPL {X  -149.536, Y  +728.383, Z    +0.000, E1   -71.359, E3 +130191.154}
SPL {X  -146.250, Y  +736.367, Z    +0.000, E1   -70.965, E3 +130199.709}
SPL {X  -143.481, Y  +742.281, Z    +0.000, E1   -70.623, E3 +130206.304}
SPL {X  -140.071, Y  +748.811, Z    +0.000, E1   -70.193, E3 +130213.816}
SPL {X  -136.578, Y  +754.826, Z    +0.000, E1   -69.723, E3 +130220.945}
SPL {X  -133.265, Y  +760.028, Z    +0.000, E1   -69.258, E3 +130227.246}
SPL {X  -130.837, Y  +763.579, Z    +0.000, E1   -68.898, E3 +130231.606}
SPL {X  -127.941, Y  +767.561, Z    +0.000, E1   -68.475, E3 +130236.496}
SPL {X  -123.778, Y  +772.869, Z    +0.000, E1   -67.843, E3 +130243.004}
SPL {X   -84.435, Y  +807.395, Z    +0.000, E1   -55.948, E3 +130355.743}
ENDSPLINE

SPLINE
SPL {X  -119.703, Y  +777.650, Z    +0.000, E1   -51.831, E3 +130519.750}
SPL {X  -145.184, Y  +738.720, Z    +0.000, E1   -43.488, E3 +130546.308}
SPL {X  -154.467, Y  +713.173, Z    +0.000, E1   -32.658, E3 +130553.903}
SPL {X  -157.530, Y  +699.446, Z    +0.000, E1   -24.482, E3 +130556.319}
SPL {X  -159.337, Y  +685.942, Z    +0.000, E1   -14.672, E3 +130557.744}
SPL {X  -159.900, Y  +676.871, Z    +0.000, E1    -6.955, E3 +130558.292}
SPL {X  -159.990, Y  +669.634, Z    +0.000, E1    -0.285, E3 +130558.435}
SPL {X  -159.990, Y  +667.035, Z    +0.000, E1    +4.539, E3 +130558.467}
SPL {X  -159.990, Y  +662.914, Z    +0.000, E1   +13.494, E3 +130558.606}
SPL {X  -159.990, Y  +658.254, Z    +0.000, E1   +24.153, E3 +130558.884}
SPL {X  -159.990, Y  +652.944, Z    +0.000, E1   +35.122, E3 +130559.387}
SPL {X  -159.990, Y  +646.557, Z    +0.000, E1   +45.390, E3 +130560.254}
SPL {X  -159.990, Y  +638.701, Z    +0.000, E1   +53.953, E3 +130561.621}
SPL {X  -159.990, Y  +618.566, Z    +0.000, E1   +64.119, E3 +130567.130}
SPL {X  -159.990, Y  +582.261, Z    +0.000, E1   +69.343, E3 +130580.615}
SPL {X  -159.990, Y  +406.555, Z    +0.000, E1   +71.635, E3 +130676.862}
SPL {X  -159.967, Y  +379.776, Z    +0.000, E1   +71.634, E3 +130695.755}
SPL {X  -158.535, Y  +360.970, Z    +0.000, E1   +71.460, E3 +130710.577}
SPL {X  -156.277, Y  +348.230, Z    +0.000, E1   +71.211, E3 +130721.920}
SPL {X  -155.351, Y  +344.251, Z    +0.000, E1   +70.004, E3 +130735.712}
SPL {X  -150.579, Y  +328.438, Z    +0.000, E1   +70.374, E3 +130744.097}
SPL {X  -146.933, Y  +319.195, Z    +0.000, E1   +70.230, E3 +130751.788}
SPL {X  -143.573, Y  +311.906, Z    +0.000, E1   +69.806, E3 +130760.099}
SPL {X  -140.547, Y  +306.057, Z    +0.000, E1   +69.399, E3 +130766.991}
SPL {X  -137.438, Y  +300.600, Z    +0.000, E1   +68.984, E3 +130773.585}
SPL {X  -133.397, Y  +294.172, Z    +0.000, E1   +68.416, E3 +130781.520}
SPL {X  -129.981, Y  +289.217, Z    +0.000, E1   +67.880, E3 +130787.769}
SPL {X  -126.457, Y  +284.492, Z    +0.000, E1   +67.352, E3 +130793.706}
SPL {X  -123.432, Y  +280.710, Z    +0.000, E1   +66.830, E3 +130798.492}
SPL {X   -85.607, Y  +247.340, Z    +0.000, E1   +53.917, E3 +130940.213}
ENDSPLINE

SPLINE
SPL {X  -119.557, Y  +276.184, Z    +0.000, E1   +51.032, E3 +131063.749}
SPL {X  -138.294, Y  +302.054, Z    +0.000, E1   +46.576, E3 +131087.072}
SPL {X  -153.211, Y  +336.421, Z    +0.000, E1   +34.262, E3 +131100.194}
SPL {X  -158.240, Y  +358.900, Z    +0.000, E1   +21.089, E3 +131104.399}
SPL {X  -159.674, Y  +372.451, Z    +0.000, E1   +10.778, E3 +131105.695}
SPL {X  -159.987, Y  +381.470, Z    +0.000, E1    +2.976, E3 +131106.052}
SPL {X  -159.990, Y  +384.761, Z    +0.000, E1    -0.257, E3 +131106.087}
SPL {X  -159.990, Y  +389.248, Z    +0.000, E1    -8.879, E3 +131106.191}
SPL {X  -159.990, Y  +394.559, Z    +0.000, E1   -20.770, E3 +131106.490}
SPL {X  -159.990, Y  +399.334, Z    +0.000, E1   -30.876, E3 +131106.929}
SPL {X  -159.990, Y  +405.006, Z    +0.000, E1   -40.810, E3 +131107.646}
SPL {X  -159.990, Y  +415.193, Z    +0.000, E1   -52.724, E3 +131109.534}
SPL {X  -159.990, Y  +465.395, Z    +0.000, E1   -68.959, E3 +131124.622}
SPL {X  -159.990, Y  +657.157, Z    +0.000, E1   -72.499, E3 +131221.019}
SPL {X  -159.693, Y  +681.249, Z    +0.000, E1   -72.488, E3 +131237.413}
SPL {X  -157.599, Y  +699.059, Z    +0.000, E1   -72.249, E3 +131251.573}
SPL {X  -155.217, Y  +710.289, Z    +0.000, E1   -71.989, E3 +131261.589}
SPL {X  -152.611, Y  +719.527, Z    +0.000, E1   -71.702, E3 +131270.410}
SPL {X  -149.536, Y  +728.383, Z    +0.000, E1   -71.359, E3 +131279.390}
SPL {X  -146.250, Y  +736.367, Z    +0.000, E1   -70.965, E3 +131287.944}
SPL {X  -143.481, Y  +742.281, Z    +0.000, E1   -70.623, E3 +131294.539}
SPL {X  -140.071, Y  +748.811, Z    +0.000, E1   -70.193, E3 +131302.051}
SPL {X  -136.578, Y  +754.826, Z    +0.000, E1   -69.723, E3 +131309.180}
SPL {X  -133.265, Y  +760.028, Z    +0.000, E1   -69.258, E3 +131315.481}
SPL {X  -129.890, Y  +764.909, Z    +0.000, E1   -68.775, E3 +131321.452}
SPL {X  -125.802, Y  +770.346, Z    +0.000, E1   -68.156, E3 +131328.151}
SPL {X  -122.624, Y  +774.263, Z    +0.000, E1   -67.622, E3 +131332.974}
SPL {X   -84.435, Y  +807.395, Z    +0.000, E1   -55.948, E3 +131443.978}
ENDSPLINE

SPLINE
SPL {X  -119.703, Y  +777.650, Z    +0.000, E1   -51.831, E3 +131607.985}
SPL {X  -145.184, Y  +738.720, Z    +0.000, E1   -43.488, E3 +131634.543}
SPL {X  -156.175, Y  +706.232, Z    +0.000, E1   -28.819, E3 +131643.428}
SPL {X  -159.337, Y  +685.942, Z    +0.000, E1   -14.672, E3 +131645.979}
SPL {X  -159.900, Y  +676.871, Z    +0.000, E1    -6.955, E3 +131646.527}
SPL {X  -159.990, Y  +669.634, Z    +0.000, E1    -0.285, E3 +131646.670}
SPL {X  -159.990, Y  +667.035, Z    +0.000, E1    +4.539, E3 +131646.702}
SPL {X  -159.990, Y  +662.914, Z    +0.000, E1   +13.494, E3 +131646.841}
SPL {X  -159.990, Y  +658.254, Z    +0.000, E1   +24.153, E3 +131647.119}
SPL {X  -159.990, Y  +652.944, Z    +0.000, E1   +35.122, E3 +131647.623}
SPL {X  -159.990, Y  +646.557, Z    +0.000, E1   +45.390, E3 +131648.490}
SPL {X  -159.990, Y  +638.701, Z    +0.000, E1   +53.953, E3 +131649.857}
SPL {X  -159.990, Y  +618.566, Z    +0.000, E1   +64.119, E3 +131655.365}
SPL {X  -159.990, Y  +582.261, Z    +0.000, E1   +69.343, E3 +131668.851}
SPL {X  -159.990, Y  +414.423, Z    +0.000, E1   +71.602, E3 +131759.634}
SPL {X  -159.990, Y  +400.357, Z    +0.000, E1   +71.604, E3 +131769.545}
SPL {X  -159.990, Y  +385.723, Z    +0.000, E1   +71.610, E3 +131779.835}
SPL {X  -159.404, Y  +368.814, Z    +0.000, E1   +71.556, E3 +131792.365}
SPL {X  -157.440, Y  +354.048, Z    +0.000, E1   +71.342, E3 +131804.838}
SPL {X  -155.889, Y  +346.508, Z    +0.000, E1   +70.461, E3 +131818.386}
SPL {X  -154.332, Y  +340.328, Z    +0.000, E1   +70.024, E3 +131826.614}
SPL {X  -150.579, Y  +328.438, Z    +0.000, E1   +70.374, E3 +131832.333}
SPL {X  -146.933, Y  +319.195, Z    +0.000, E1   +70.230, E3 +131840.024}
SPL {X  -143.573, Y  +311.906, Z    +0.000, E1   +69.806, E3 +131848.334}
SPL {X  -139.693, Y  +304.508, Z    +0.000, E1   +69.301, E3 +131857.062}
SPL {X  -135.622, Y  +297.627, Z    +0.000, E1   +68.731, E3 +131865.470}
SPL {X  -132.531, Y  +292.877, Z    +0.000, E1   +68.266, E3 +131871.406}
SPL {X  -128.822, Y  +287.623, Z    +0.000, E1   +67.729, E3 +131877.980}
SPL {X  -124.502, Y  +282.021, Z    +0.000, E1   +67.035, E3 +131885.054}
SPL {X   -85.607, Y  +247.340, Z    +0.000, E1   +53.917, E3 +132028.448}
ENDSPLINE

SPLINE
SPL {X  -134.737, Y  +296.229, Z    +0.000, E1   +47.890, E3 +132171.221}
SPL {X  -153.211, Y  +336.421, Z    +0.000, E1   +34.262, E3 +132188.429}
SPL {X  -158.240, Y  +358.900, Z    +0.000, E1   +21.089, E3 +132192.634}
SPL {X  -159.674, Y  +372.451, Z    +0.000, E1   +10.778, E3 +132193.930}
SPL {X  -159.987, Y  +381.470, Z    +0.000, E1    +2.976, E3 +132194.287}
SPL {X  -159.990, Y  +384.761, Z    +0.000, E1    -0.257, E3 +132194.322}
SPL {X  -159.990, Y  +389.248, Z    +0.000, E1    -8.879, E3 +132194.426}
SPL {X  -159.990, Y  +394.559, Z    +0.000, E1   -20.770, E3 +132194.725}
SPL {X  -159.990, Y  +399.334, Z    +0.000, E1   -30.876, E3 +132195.164}
SPL {X  -159.990, Y  +405.006, Z    +0.000, E1   -40.810, E3 +132195.882}
SPL {X  -159.990, Y  +415.193, Z    +0.000, E1   -52.724, E3 +132197.769}
SPL {X  -159.990, Y  +465.395, Z    +0.000, E1   -68.959, E3 +132212.857}
SPL {X  -159.990, Y  +657.157, Z    +0.000, E1   -72.499, E3 +132309.254}
SPL {X  -159.947, Y  +675.227, Z    +0.000, E1   -72.487, E3 +132321.414}
SPL {X  -159.251, Y  +686.856, Z    +0.000, E1   -72.412, E3 +132329.943}
SPL {X  -157.599, Y  +699.059, Z    +0.000, E1   -72.249, E3 +132339.808}
SPL {X  -155.217, Y  +710.289, Z    +0.000, E1   -71.989, E3 +132349.825}
SPL {X  -152.611, Y  +719.527, Z    +0.000, E1   -71.702, E3 +132358.646}
SPL {X  -149.536, Y  +728.383, Z    +0.000, E1   -71.359, E3 +132367.625}
SPL {X  -146.250, Y  +736.367, Z    +0.000, E1   -70.965, E3 +132376.179}
SPL {X  -143.481, Y  +742.281, Z    +0.000, E1   -70.623, E3 +132382.775}
SPL {X  -140.071, Y  +748.811, Z    +0.000, E1   -70.193, E3 +132390.286}
SPL {X  -136.578, Y  +754.826, Z    +0.000, E1   -69.723, E3 +132397.416}
SPL {X  -133.265, Y  +760.028, Z    +0.000, E1   -69.258, E3 +132403.717}
SPL {X  -129.890, Y  +764.909, Z    +0.000, E1   -68.775, E3 +132409.687}
SPL {X  -125.802, Y  +770.346, Z    +0.000, E1   -68.156, E3 +132416.386}
SPL {X  -122.624, Y  +774.263, Z    +0.000, E1   -67.622, E3 +132421.209}
SPL {X   -84.435, Y  +807.395, Z    +0.000, E1   -55.948, E3 +132532.214}
ENDSPLINE

SPLINE
SPL {X  -119.703, Y  +777.650, Z    +0.000, E1   -51.831, E3 +132696.220}
SPL {X  -145.184, Y  +738.720, Z    +0.000, E1   -43.488, E3 +132722.778}
SPL {X  -156.175, Y  +706.232, Z    +0.000, E1   -28.819, E3 +132731.663}
SPL {X  -159.337, Y  +685.942, Z    +0.000, E1   -14.672, E3 +132734.214}
SPL {X  -159.962, Y  +674.468, Z    +0.000, E1    -4.846, E3 +132734.833}
SPL {X  -159.990, Y  +669.479, Z    +0.000, E1    +0.004, E3 +132734.907}
SPL {X  -159.990, Y  +667.035, Z    +0.000, E1    +4.539, E3 +132734.938}
SPL {X  -159.990, Y  +662.914, Z    +0.000, E1   +13.494, E3 +132735.077}
SPL {X  -159.990, Y  +658.254, Z    +0.000, E1   +24.153, E3 +132735.354}
SPL {X  -159.990, Y  +652.944, Z    +0.000, E1   +35.122, E3 +132735.858}
SPL {X  -159.990, Y  +642.509, Z    +0.000, E1   +50.090, E3 +132737.430}
SPL {X  -159.990, Y  +618.566, Z    +0.000, E1   +64.119, E3 +132743.600}
SPL {X  -159.990, Y  +582.261, Z    +0.000, E1   +69.343, E3 +132757.086}
SPL {X  -159.990, Y  +406.555, Z    +0.000, E1   +71.635, E3 +132853.332}
SPL {X  -159.990, Y  +385.723, Z    +0.000, E1   +71.610, E3 +132868.071}
SPL {X  -159.404, Y  +368.814, Z    +0.000, E1   +71.556, E3 +132880.600}
SPL {X  -157.440, Y  +354.048, Z    +0.000, E1   +71.342, E3 +132893.073}
SPL {X  -155.538, Y  +345.018, Z    +0.000, E1   +71.109, E3 +132901.466}
SPL {X  -155.351, Y  +344.251, Z    +0.000, E1   +70.004, E3 +132912.183}
SPL {X  -150.579, Y  +328.438, Z    +0.000, E1   +70.374, E3 +132920.568}
SPL {X  -146.933, Y  +319.195, Z    +0.000, E1   +70.230, E3 +132928.259}
SPL {X  -143.573, Y  +311.906, Z    +0.000, E1   +69.806, E3 +132936.569}
SPL {X  -140.547, Y  +306.057, Z    +0.000, E1   +69.399, E3 +132943.461}
SPL {X  -137.438, Y  +300.600, Z    +0.000, E1   +68.984, E3 +132950.056}
SPL {X  -133.397, Y  +294.172, Z    +0.000, E1   +68.416, E3 +132957.990}
SPL {X  -128.822, Y  +287.623, Z    +0.000, E1   +67.729, E3 +132966.215}
SPL {X  -124.502, Y  +282.021, Z    +0.000, E1   +67.035, E3 +132973.289}
SPL {X   -85.607, Y  +247.340, Z    +0.000, E1   +53.917, E3 +133116.683}
ENDSPLINE

SPLINE
SPL {X  -134.737, Y  +296.229, Z    +0.000, E1   +47.890, E3 +133259.456}
SPL {X  -154.917, Y  +342.531, Z    +0.000, E1   +31.203, E3 +133278.024}
SPL {X  -159.440, Y  +369.246, Z    +0.000, E1   +13.458, E3 +133281.923}
SPL {X  -159.957, Y  +379.264, Z    +0.000, E1    +4.909, E3 +133282.479}
SPL {X  -159.990, Y  +384.670, Z    +0.000, E1    -0.079, E3 +133282.557}
SPL {X  -159.990, Y  +389.248, Z    +0.000, E1    -8.879, E3 +133282.661}
SPL {X  -159.990, Y  +394.559, Z    +0.000, E1   -20.770, E3 +133282.960}
SPL {X  -159.990, Y  +399.334, Z    +0.000, E1   -30.876, E3 +133283.399}
SPL {X  -159.990, Y  +405.006, Z    +0.000, E1   -40.810, E3 +133284.117}
SPL {X  -159.990, Y  +415.193, Z    +0.000, E1   -52.724, E3 +133286.004}
SPL {X  -159.990, Y  +465.395, Z    +0.000, E1   -68.959, E3 +133301.093}
SPL {X  -159.990, Y  +657.157, Z    +0.000, E1   -72.499, E3 +133397.490}
SPL {X  -159.693, Y  +681.249, Z    +0.000, E1   -72.488, E3 +133413.884}
SPL {X  -157.599, Y  +699.059, Z    +0.000, E1   -72.249, E3 +133428.043}
SPL {X  -155.217, Y  +710.289, Z    +0.000, E1   -71.989, E3 +133438.060}
SPL {X  -152.611, Y  +719.527, Z    +0.000, E1   -71.702, E3 +133446.881}
SPL {X  -149.536, Y  +728.383, Z    +0.000, E1   -71.359, E3 +133455.860}
SPL {X  -146.250, Y  +736.367, Z    +0.000, E1   -70.965, E3 +133464.414}
SPL {X  -143.481, Y  +742.281, Z    +0.000, E1   -70.623, E3 +133471.010}
SPL {X  -140.071, Y  +748.811, Z    +0.000, E1   -70.193, E3 +133478.522}
SPL {X  -136.578, Y  +754.826, Z    +0.000, E1   -69.723, E3 +133485.651}
SPL {X  -133.265, Y  +760.028, Z    +0.000, E1   -69.258, E3 +133491.952}
SPL {X  -129.890, Y  +764.909, Z    +0.000, E1   -68.775, E3 +133497.923}
SPL {X  -125.802, Y  +770.346, Z    +0.000, E1   -68.156, E3 +133504.622}
SPL {X  -122.624, Y  +774.263, Z    +0.000, E1   -67.622, E3 +133509.444}
SPL {X   -84.435, Y  +807.395, Z    +0.000, E1   -55.948, E3 +133620.449}
ENDSPLINE

SPLINE
SPL {X  -119.703, Y  +777.650, Z    +0.000, E1   -51.831, E3 +133784.455}
SPL {X  -145.184, Y  +738.720, Z    +0.000, E1   -43.488, E3 +133811.013}
SPL {X  -154.467, Y  +713.173, Z    +0.000, E1   -32.658, E3 +133818.609}
SPL {X  -157.530, Y  +699.446, Z    +0.000, E1   -24.482, E3 +133821.025}
SPL {X  -159.337, Y  +685.942, Z    +0.000, E1   -14.672, E3 +133822.449}
SPL {X  -159.900, Y  +676.871, Z    +0.000, E1    -6.955, E3 +133822.998}
SPL {X  -159.990, Y  +669.634, Z    +0.000, E1    -0.285, E3 +133823.141}
SPL {X  -159.990, Y  +667.035, Z    +0.000, E1    +4.539, E3 +133823.173}
SPL {X  -159.990, Y  +662.914, Z    +0.000, E1   +13.494, E3 +133823.312}
SPL {X  -159.990, Y  +658.254, Z    +0.000, E1   +24.153, E3 +133823.590}
SPL {X  -159.990, Y  +652.944, Z    +0.000, E1   +35.122, E3 +133824.093}
SPL {X  -159.990, Y  +642.509, Z    +0.000, E1   +50.090, E3 +133825.665}
SPL {X  -159.990, Y  +618.566, Z    +0.000, E1   +64.119, E3 +133831.835}
SPL {X  -159.990, Y  +582.261, Z    +0.000, E1   +69.343, E3 +133845.321}
SPL {X  -159.990, Y  +406.555, Z    +0.000, E1   +71.635, E3 +133941.568}
SPL {X  -159.990, Y  +385.723, Z    +0.000, E1   +71.610, E3 +133956.306}
SPL {X  -159.404, Y  +368.814, Z    +0.000, E1   +71.556, E3 +133968.835}
SPL {X  -158.061, Y  +357.731, Z    +0.000, E1   +71.393, E3 +133978.103}
SPL {X  -156.277, Y  +348.230, Z    +0.000, E1   +71.211, E3 +133986.626}
SPL {X  -155.351, Y  +344.251, Z    +0.000, E1   +70.004, E3 +134000.418}
SPL {X  -150.579, Y  +328.438, Z    +0.000, E1   +70.374, E3 +134008.803}
SPL {X  -146.933, Y  +319.195, Z    +0.000, E1   +70.230, E3 +134016.494}
SPL {X  -143.573, Y  +311.906, Z    +0.000, E1   +69.806, E3 +134024.805}
SPL {X  -140.547, Y  +306.057, Z    +0.000, E1   +69.399, E3 +134031.696}
SPL {X  -136.400, Y  +298.883, Z    +0.000, E1   +68.867, E3 +134040.352}
SPL {X  -131.165, Y  +290.889, Z    +0.000, E1   +68.094, E3 +134050.326}
SPL {X  -126.457, Y  +284.492, Z    +0.000, E1   +67.352, E3 +134058.412}
SPL {X  -123.432, Y  +280.710, Z    +0.000, E1   +66.830, E3 +134063.197}
SPL {X   -85.607, Y  +247.340, Z    +0.000, E1   +53.917, E3 +134204.919}
ENDSPLINE

SPLINE
SPL {X  -134.737, Y  +296.229, Z    +0.000, E1   +47.890, E3 +134347.692}
SPL {X  -154.917, Y  +342.531, Z    +0.000, E1   +31.203, E3 +134366.259}
SPL {X  -159.440, Y  +369.246, Z    +0.000, E1   +13.458, E3 +134370.159}
SPL {X  -159.987, Y  +381.470, Z    +0.000, E1    +2.976, E3 +134370.757}
SPL {X  -159.990, Y  +384.761, Z    +0.000, E1    -0.257, E3 +134370.793}
SPL {X  -159.990, Y  +389.248, Z    +0.000, E1    -8.879, E3 +134370.896}
SPL {X  -159.990, Y  +394.559, Z    +0.000, E1   -20.770, E3 +134371.195}
SPL {X  -159.990, Y  +399.334, Z    +0.000, E1   -30.876, E3 +134371.634}
SPL {X  -159.990, Y  +405.006, Z    +0.000, E1   -40.810, E3 +134372.352}
SPL {X  -159.990, Y  +415.193, Z    +0.000, E1   -52.724, E3 +134374.239}
SPL {X  -159.990, Y  +465.395, Z    +0.000, E1   -68.959, E3 +134389.328}
SPL {X  -159.990, Y  +657.157, Z    +0.000, E1   -72.499, E3 +134485.725}
SPL {X  -159.693, Y  +681.249, Z    +0.000, E1   -72.488, E3 +134502.119}
SPL {X  -157.599, Y  +699.059, Z    +0.000, E1   -72.249, E3 +134516.278}
SPL {X  -155.217, Y  +710.289, Z    +0.000, E1   -71.989, E3 +134526.295}
SPL {X  -152.611, Y  +719.527, Z    +0.000, E1   -71.702, E3 +134535.116}
SPL {X  -149.536, Y  +728.383, Z    +0.000, E1   -71.359, E3 +134544.096}
SPL {X  -146.250, Y  +736.367, Z    +0.000, E1   -70.965, E3 +134552.650}
SPL {X  -143.481, Y  +742.281, Z    +0.000, E1   -70.623, E3 +134559.245}
SPL {X  -140.071, Y  +748.811, Z    +0.000, E1   -70.193, E3 +134566.757}
SPL {X  -136.578, Y  +754.826, Z    +0.000, E1   -69.723, E3 +134573.886}
SPL {X  -133.265, Y  +760.028, Z    +0.000, E1   -69.258, E3 +134580.187}
SPL {X  -129.890, Y  +764.909, Z    +0.000, E1   -68.775, E3 +134586.158}
SPL {X  -125.802, Y  +770.346, Z    +0.000, E1   -68.156, E3 +134592.857}
SPL {X  -122.624, Y  +774.263, Z    +0.000, E1   -67.622, E3 +134597.680}
SPL {X   -84.435, Y  +807.395, Z    +0.000, E1   -55.948, E3 +134708.684}
ENDSPLINE

SPLINE
SPL {X  -119.703, Y  +777.650, Z    +0.000, E1   -51.831, E3 +134872.691}
SPL {X  -145.184, Y  +738.720, Z    +0.000, E1   -43.488, E3 +134899.249}
SPL {X  -154.467, Y  +713.173, Z    +0.000, E1   -32.658, E3 +134906.844}
SPL {X  -157.530, Y  +699.446, Z    +0.000, E1   -24.482, E3 +134909.260}
SPL {X  -159.337, Y  +685.942, Z    +0.000, E1   -14.672, E3 +134910.685}
SPL {X  -159.962, Y  +674.468, Z    +0.000, E1    -4.846, E3 +134911.303}
SPL {X  -159.990, Y  +669.479, Z    +0.000, E1    +0.004, E3 +134911.378}
SPL {X  -159.990, Y  +667.035, Z    +0.000, E1    +4.539, E3 +134911.408}
SPL {X  -159.990, Y  +662.914, Z    +0.000, E1   +13.494, E3 +134911.547}
SPL {X  -159.990, Y  +658.254, Z    +0.000, E1   +24.153, E3 +134911.825}
SPL {X  -159.990, Y  +652.944, Z    +0.000, E1   +35.122, E3 +134912.329}
SPL {X  -159.990, Y  +642.509, Z    +0.000, E1   +50.090, E3 +134913.900}
SPL {X  -159.990, Y  +618.566, Z    +0.000, E1   +64.119, E3 +134920.071}
SPL {X  -159.990, Y  +582.261, Z    +0.000, E1   +69.343, E3 +134933.556}
SPL {X  -159.990, Y  +406.555, Z    +0.000, E1   +71.635, E3 +135029.803}
SPL {X  -159.990, Y  +385.723, Z    +0.000, E1   +71.610, E3 +135044.541}
SPL {X  -159.404, Y  +368.814, Z    +0.000, E1   +71.556, E3 +135057.071}
SPL {X  -158.061, Y  +357.731, Z    +0.000, E1   +71.393, E3 +135066.338}
SPL {X  -156.277, Y  +348.230, Z    +0.000, E1   +71.211, E3 +135074.861}
SPL {X  -155.351, Y  +344.251, Z    +0.000, E1   +70.004, E3 +135088.653}
SPL {X  -150.579, Y  +328.438, Z    +0.000, E1   +70.374, E3 +135097.039}
SPL {X  -146.933, Y  +319.195, Z    +0.000, E1   +70.230, E3 +135104.730}
SPL {X  -143.573, Y  +311.906, Z    +0.000, E1   +69.806, E3 +135113.040}
SPL {X  -140.547, Y  +306.057, Z    +0.000, E1   +69.399, E3 +135119.932}
SPL {X  -137.438, Y  +300.600, Z    +0.000, E1   +68.984, E3 +135126.526}
SPL {X  -133.397, Y  +294.172, Z    +0.000, E1   +68.416, E3 +135134.461}
SPL {X  -129.981, Y  +289.217, Z    +0.000, E1   +67.880, E3 +135140.711}
SPL {X  -126.457, Y  +284.492, Z    +0.000, E1   +67.352, E3 +135146.647}
SPL {X  -123.432, Y  +280.710, Z    +0.000, E1   +66.830, E3 +135151.433}
SPL {X   -85.607, Y  +247.340, Z    +0.000, E1   +53.917, E3 +135293.154}
ENDSPLINE

